Yaskawa INFORM job: DEMO_ROOF_SIDE_0625_3PAINT_39.JBI

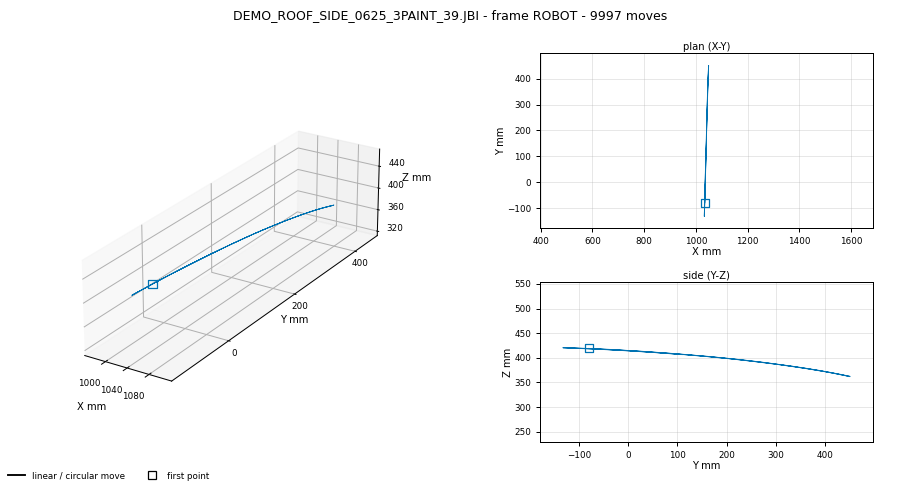
[picture p0: tool path of DEMO_ROOF_SIDE_0625_3PAINT_39.JBI in frame ROBOT, 9997 of 9997 moves have a stored position in this frame; points joined in program order, loops and branches not executed]
/JOB
//NAME DEMO_ROOF_SIDE_0625_3PAINT39
//POS
///NPOS 9997,0,0,0,0,0
///TOOL 0
///USER 0
///POSTYPE ROBOT
///RECTAN
///RCONF 1,0,0,0,0,0,0,0,0,0,0,0,0,0,0,0,0,0,0,0,0,0,0,0
C00000=1034.814,-80.144,419.319,168.128,39.375,157.359
C00001=1034.820,-79.894,419.308,168.131,39.374,157.359
C00002=1034.826,-79.644,419.297,168.134,39.373,157.359
C00003=1034.832,-79.394,419.285,168.136,39.372,157.359
C00004=1034.838,-79.144,419.275,168.139,39.372,157.359
C00005=1034.844,-78.895,419.264,168.142,39.371,157.359
C00006=1034.851,-78.645,419.253,168.144,39.371,157.359
C00007=1034.856,-78.396,419.242,168.147,39.370,157.358
C00008=1034.863,-78.145,419.231,168.150,39.369,157.358
C00009=1034.868,-77.896,419.220,168.152,39.368,157.358
C00010=1034.875,-77.646,419.209,168.155,39.368,157.358
C00011=1034.881,-77.397,419.197,168.157,39.367,157.358
C00012=1034.886,-77.147,419.186,168.160,39.366,157.358
C00013=1034.893,-76.897,419.175,168.162,39.365,157.358
C00014=1034.899,-76.648,419.164,168.165,39.364,157.358
C00015=1034.906,-76.398,419.154,168.168,39.364,157.358
C00016=1034.911,-76.148,419.143,168.170,39.363,157.358
C00017=1034.918,-75.899,419.131,168.173,39.362,157.358
C00018=1034.924,-75.649,419.120,168.176,39.361,157.358
C00019=1034.930,-75.399,419.109,168.179,39.361,157.358
C00020=1034.936,-75.150,419.098,168.181,39.360,157.358
C00021=1034.942,-74.899,419.086,168.184,39.360,157.358
C00022=1034.948,-74.650,419.075,168.187,39.359,157.358
C00023=1034.955,-74.400,419.064,168.189,39.358,157.358
C00024=1034.960,-74.151,419.053,168.192,39.358,157.358
C00025=1034.967,-73.901,419.041,168.195,39.357,157.358
C00026=1034.973,-73.652,419.030,168.196,39.356,157.358
C00027=1034.979,-73.402,419.019,168.199,39.356,157.358
C00028=1034.985,-73.153,419.007,168.202,39.355,157.358
C00029=1034.991,-72.902,418.995,168.204,39.355,157.358
C00030=1034.996,-72.653,418.984,168.207,39.354,157.358
C00031=1035.002,-72.404,418.973,168.210,39.354,157.358
C00032=1035.009,-72.154,418.962,168.212,39.353,157.358
C00033=1035.015,-71.904,418.951,168.215,39.352,157.358
C00034=1035.020,-71.654,418.938,168.217,39.352,157.358
C00035=1035.027,-71.404,418.927,168.220,39.351,157.358
C00036=1035.033,-71.155,418.915,168.223,39.351,157.358
C00037=1035.039,-70.905,418.904,168.225,39.350,157.358
C00038=1035.045,-70.656,418.893,168.228,39.350,157.358
C00039=1035.051,-70.406,418.881,168.231,39.349,157.358
C00040=1035.057,-70.156,418.870,168.233,39.348,157.357
C00041=1035.063,-69.907,418.858,168.236,39.348,157.357
C00042=1035.069,-69.657,418.847,168.239,39.347,157.357
C00043=1035.076,-69.408,418.835,168.241,39.347,157.357
C00044=1035.081,-69.158,418.823,168.244,39.346,157.357
C00045=1035.087,-68.908,418.812,168.246,39.346,157.357
C00046=1035.094,-68.658,418.800,168.249,39.345,157.357
C00047=1035.100,-68.375,418.787,168.251,39.344,157.357
C00048=1035.107,-68.093,418.774,168.254,39.344,157.357
C00049=1035.114,-67.811,418.761,168.257,39.343,157.357
C00050=1035.121,-67.528,418.748,168.260,39.342,157.357
C00051=1035.127,-67.278,418.736,168.263,39.342,157.357
C00052=1035.133,-67.028,418.724,168.265,39.341,157.357
C00053=1035.139,-66.778,418.713,168.268,39.341,157.357
C00054=1035.145,-66.529,418.701,168.271,39.340,157.357
C00055=1035.152,-66.279,418.690,168.273,39.340,157.357
C00056=1035.157,-66.029,418.677,168.276,39.339,157.357
C00057=1035.164,-65.780,418.666,168.278,39.339,157.357
C00058=1035.170,-65.530,418.655,168.281,39.338,157.357
C00059=1035.176,-65.281,418.643,168.284,39.337,157.357
C00060=1035.182,-65.030,418.631,168.286,39.337,157.357
C00061=1035.188,-64.781,418.619,168.289,39.336,157.357
C00062=1035.194,-64.532,418.607,168.292,39.336,157.357
C00063=1035.201,-64.282,418.596,168.294,39.335,157.357
C00064=1035.206,-64.032,418.584,168.297,39.335,157.357
C00065=1035.213,-63.783,418.572,168.299,39.334,157.357
C00066=1035.219,-63.533,418.561,168.302,39.334,157.357
C00067=1035.226,-63.283,418.549,168.305,39.333,157.357
C00068=1035.231,-63.034,418.537,168.307,39.333,157.357
C00069=1035.237,-62.784,418.525,168.310,39.332,157.357
C00070=1035.244,-62.534,418.513,168.311,39.331,157.357
C00071=1035.250,-62.285,418.502,168.314,39.331,157.357
C00072=1035.256,-62.035,418.489,168.317,39.330,157.357
C00073=1035.262,-61.785,418.478,168.319,39.330,157.357
C00074=1035.269,-61.536,418.466,168.322,39.329,157.357
C00075=1035.274,-61.286,418.454,168.324,39.329,157.357
C00076=1035.281,-61.037,418.442,168.327,39.328,157.357
C00077=1035.287,-60.787,418.431,168.330,39.327,157.357
C00078=1035.294,-60.537,418.419,168.332,39.327,157.357
C00079=1035.299,-60.288,418.406,168.335,39.326,157.357
C00080=1035.306,-60.038,418.394,168.338,39.326,157.357
C00081=1035.312,-59.788,418.383,168.340,39.325,157.357
C00082=1035.318,-59.538,418.371,168.343,39.325,157.357
C00083=1035.325,-59.289,418.359,168.345,39.324,157.357
C00084=1035.331,-59.040,418.347,168.348,39.324,157.357
C00085=1035.337,-58.790,418.335,168.351,39.323,157.357
C00086=1035.343,-58.540,418.323,168.353,39.322,157.357
C00087=1035.350,-58.290,418.311,168.356,39.322,157.357
C00088=1035.356,-58.041,418.299,168.358,39.321,157.357
C00089=1035.362,-57.791,418.287,168.361,39.321,157.357
C00090=1035.368,-57.542,418.275,168.364,39.320,157.357
C00091=1035.375,-57.292,418.263,168.366,39.320,157.357
C00092=1035.381,-57.042,418.251,168.369,39.319,157.357
C00093=1035.388,-56.793,418.239,168.371,39.319,157.357
C00094=1035.394,-56.543,418.227,168.374,39.318,157.357
C00095=1035.401,-56.294,418.215,168.375,39.318,157.357
C00096=1035.406,-56.044,418.203,168.378,39.317,157.357
C00097=1035.412,-55.794,418.191,168.381,39.316,157.357
C00098=1035.419,-55.545,418.179,168.383,39.316,157.357
C00099=1035.425,-55.295,418.167,168.386,39.315,157.357
C00100=1035.432,-55.045,418.155,168.388,39.315,157.357
C00101=1035.438,-54.796,418.143,168.391,39.314,157.357
C00102=1035.444,-54.546,418.130,168.394,39.313,157.357
C00103=1035.451,-54.296,418.118,168.396,39.313,157.357
C00104=1035.458,-54.047,418.107,168.399,39.312,157.357
C00105=1035.463,-53.797,418.094,168.401,39.312,157.357
C00106=1035.469,-53.548,418.082,168.404,39.311,157.356
C00107=1035.476,-53.298,418.070,168.407,39.311,157.357
C00108=1035.482,-53.048,418.058,168.409,39.310,157.356
C00109=1035.489,-52.799,418.046,168.412,39.310,157.357
C00110=1035.495,-52.549,418.034,168.414,39.309,157.356
C00111=1035.503,-52.268,418.020,168.417,39.309,157.356
C00112=1035.510,-51.986,418.006,168.420,39.308,157.356
C00113=1035.516,-51.705,417.992,168.423,39.307,157.356
C00114=1035.524,-51.423,417.979,168.426,39.307,157.356
C00115=1035.530,-51.174,417.966,168.428,39.306,157.356
C00116=1035.537,-50.924,417.954,168.431,39.306,157.356
C00117=1035.543,-50.674,417.942,168.434,39.305,157.356
C00118=1035.549,-50.424,417.930,168.436,39.305,157.356
C00119=1035.556,-50.175,417.916,168.439,39.305,157.356
C00120=1035.562,-49.926,417.904,168.440,39.304,157.356
C00121=1035.568,-49.676,417.892,168.444,39.304,157.356
C00122=1035.574,-49.426,417.879,168.446,39.304,157.356
C00123=1035.581,-49.176,417.867,168.449,39.304,157.357
C00124=1035.587,-48.927,417.854,168.450,39.303,157.356
C00125=1035.593,-48.677,417.841,168.453,39.303,157.356
C00126=1035.598,-48.428,417.829,168.456,39.302,157.357
C00127=1035.605,-48.178,417.817,168.459,39.302,157.357
C00128=1035.611,-47.929,417.804,168.460,39.301,157.356
C00129=1035.617,-47.679,417.792,168.463,39.301,157.357
C00130=1035.624,-47.430,417.780,168.465,39.301,157.357
C00131=1035.630,-47.180,417.766,168.468,39.300,157.357
C00132=1035.636,-46.931,417.754,168.470,39.300,157.357
C00133=1035.642,-46.681,417.741,168.473,39.300,157.357
C00134=1035.649,-46.432,417.729,168.475,39.300,157.357
C00135=1035.654,-46.182,417.716,168.478,39.299,157.357
C00136=1035.660,-45.932,417.703,168.480,39.299,157.357
C00137=1035.667,-45.683,417.690,168.483,39.298,157.357
C00138=1035.673,-45.433,417.678,168.485,39.298,157.357
C00139=1035.679,-45.183,417.666,168.488,39.297,157.357
C00140=1035.686,-44.933,417.652,168.490,39.297,157.357
C00141=1035.693,-44.684,417.640,168.493,39.297,157.357
C00142=1035.698,-44.434,417.627,168.495,39.297,157.357
C00143=1035.705,-44.185,417.614,168.498,39.296,157.357
C00144=1035.711,-43.935,417.602,168.500,39.296,157.357
C00145=1035.718,-43.686,417.589,168.503,39.296,157.357
C00146=1035.723,-43.436,417.576,168.505,39.295,157.357
C00147=1035.729,-43.186,417.564,168.507,39.295,157.357
C00148=1035.736,-42.937,417.551,168.510,39.294,157.357
C00149=1035.742,-42.687,417.539,168.512,39.294,157.357
C00150=1035.748,-42.438,417.525,168.515,39.293,157.357
C00151=1035.754,-42.188,417.513,168.517,39.293,157.357
C00152=1035.761,-41.939,417.500,168.520,39.293,157.357
C00153=1035.768,-41.688,417.487,168.522,39.293,157.357
C00154=1035.774,-41.439,417.474,168.525,39.292,157.357
C00155=1035.780,-41.189,417.461,168.527,39.292,157.357
C00156=1035.786,-40.940,417.448,168.530,39.292,157.357
C00157=1035.793,-40.690,417.436,168.532,39.292,157.357
C00158=1035.799,-40.441,417.423,168.535,39.291,157.357
C00159=1035.805,-40.191,417.410,168.537,39.291,157.357
C00160=1035.812,-39.941,417.397,168.540,39.290,157.357
C00161=1035.818,-39.691,417.384,168.542,39.290,157.357
C00162=1035.825,-39.442,417.371,168.545,39.289,157.357
C00163=1035.831,-39.193,417.359,168.547,39.289,157.357
C00164=1035.837,-38.943,417.346,168.550,39.289,157.357
C00165=1035.843,-38.694,417.332,168.552,39.289,157.357
C00166=1035.849,-38.443,417.319,168.554,39.288,157.357
C00167=1035.856,-38.194,417.306,168.557,39.288,157.357
C00168=1035.862,-37.944,417.294,168.559,39.288,157.357
C00169=1035.868,-37.695,417.280,168.562,39.287,157.357
C00170=1035.874,-37.446,417.267,168.564,39.287,157.357
C00171=1035.880,-37.196,417.255,168.567,39.287,157.357
C00172=1035.886,-36.947,417.241,168.569,39.287,157.357
C00173=1035.893,-36.697,417.228,168.571,39.287,157.357
C00174=1035.899,-36.447,417.214,168.574,39.287,157.357
C00175=1035.906,-36.167,417.200,168.576,39.286,157.357
C00176=1035.913,-35.885,417.185,168.579,39.286,157.357
C00177=1035.920,-35.604,417.170,168.582,39.285,157.357
C00178=1035.928,-35.323,417.156,168.585,39.285,157.358
C00179=1035.934,-35.074,417.142,168.587,39.285,157.358
C00180=1035.940,-34.824,417.129,168.589,39.285,157.358
C00181=1035.946,-34.574,417.117,168.592,39.285,157.358
C00182=1035.952,-34.325,417.103,168.594,39.284,157.358
C00183=1035.959,-34.075,417.090,168.597,39.284,157.358
C00184=1035.964,-33.826,417.076,168.599,39.284,157.358
C00185=1035.971,-33.576,417.063,168.601,39.283,157.358
C00186=1035.977,-33.326,417.050,168.604,39.283,157.358
C00187=1035.983,-33.076,417.036,168.606,39.283,157.358
C00188=1035.990,-32.827,417.023,168.609,39.283,157.358
C00189=1035.996,-32.578,417.010,168.611,39.283,157.358
C00190=1036.002,-32.329,416.997,168.614,39.282,157.358
C00191=1036.008,-32.078,416.984,168.616,39.282,157.358
C00192=1036.015,-31.829,416.970,168.618,39.282,157.358
C00193=1036.021,-31.580,416.957,168.621,39.282,157.358
C00194=1036.028,-31.330,416.943,168.623,39.281,157.358
C00195=1036.034,-31.080,416.930,168.626,39.281,157.358
C00196=1036.040,-30.831,416.917,168.628,39.281,157.358
C00197=1036.046,-30.582,416.904,168.630,39.281,157.358
C00198=1036.053,-30.332,416.890,168.633,39.280,157.358
C00199=1036.059,-30.082,416.877,168.635,39.280,157.358
C00200=1036.065,-29.833,416.864,168.637,39.280,157.358
C00201=1036.072,-29.583,416.851,168.640,39.280,157.358
C00202=1036.078,-29.333,416.837,168.643,39.280,157.358
C00203=1036.084,-29.084,416.823,168.645,39.279,157.358
C00204=1036.091,-28.834,416.810,168.647,39.279,157.358
C00205=1036.097,-28.585,416.797,168.649,39.279,157.358
C00206=1036.103,-28.335,416.783,168.652,39.278,157.358
C00207=1036.110,-28.085,416.770,168.654,39.278,157.358
C00208=1036.116,-27.836,416.756,168.658,39.278,157.359
C00209=1036.123,-27.586,416.743,168.660,39.278,157.359
C00210=1036.129,-27.337,416.729,168.662,39.278,157.359
C00211=1036.135,-27.088,416.716,168.665,39.277,157.359
C00212=1036.142,-26.838,416.703,168.667,39.277,157.359
C00213=1036.148,-26.588,416.689,168.669,39.277,157.359
C00214=1036.154,-26.339,416.675,168.672,39.277,157.359
C00215=1036.161,-26.089,416.662,168.674,39.277,157.359
C00216=1036.166,-25.839,416.648,168.676,39.277,157.359
C00217=1036.172,-25.590,416.635,168.679,39.276,157.359
C00218=1036.179,-25.341,416.620,168.681,39.276,157.359
C00219=1036.185,-25.091,416.606,168.683,39.276,157.359
C00220=1036.192,-24.841,416.593,168.686,39.276,157.359
C00221=1036.198,-24.592,416.580,168.688,39.276,157.359
C00222=1036.203,-24.342,416.566,168.690,39.276,157.359
C00223=1036.210,-24.092,416.552,168.693,39.275,157.359
C00224=1036.216,-23.843,416.539,168.695,39.275,157.359
C00225=1036.223,-23.593,416.524,168.697,39.275,157.359
C00226=1036.229,-23.344,416.511,168.700,39.275,157.359
C00227=1036.235,-23.095,416.497,168.702,39.275,157.359
C00228=1036.241,-22.845,416.483,168.704,39.275,157.359
C00229=1036.248,-22.595,416.470,168.707,39.274,157.359
C00230=1036.255,-22.346,416.455,168.709,39.274,157.359
C00231=1036.264,-21.949,416.434,168.713,39.275,157.360
C00232=1036.274,-21.552,416.412,168.716,39.274,157.360
C00233=1036.284,-21.155,416.389,168.720,39.274,157.360
C00234=1036.294,-20.758,416.368,168.724,39.274,157.360
C00235=1036.304,-20.374,416.346,168.727,39.274,157.360
C00236=1036.314,-19.990,416.325,168.731,39.273,157.360
C00237=1036.323,-19.606,416.304,168.735,39.273,157.360
C00238=1036.333,-19.222,416.282,168.738,39.273,157.360
C00239=1036.339,-18.973,416.268,168.740,39.273,157.360
C00240=1036.346,-18.723,416.255,168.743,39.272,157.360
C00241=1036.352,-18.474,416.241,168.745,39.272,157.360
C00242=1036.358,-18.224,416.227,168.747,39.272,157.360
C00243=1036.365,-17.975,416.213,168.750,39.272,157.360
C00244=1036.371,-17.725,416.198,168.753,39.272,157.360
C00245=1036.377,-17.476,416.185,168.755,39.272,157.360
C00246=1036.384,-17.226,416.171,168.758,39.271,157.360
C00247=1036.390,-16.977,416.157,168.760,39.271,157.361
C00248=1036.397,-16.727,416.143,168.762,39.271,157.361
C00249=1036.403,-16.477,416.128,168.765,39.271,157.361
C00250=1036.409,-16.228,416.115,168.767,39.271,157.361
C00251=1036.416,-15.979,416.101,168.769,39.271,157.361
C00252=1036.422,-15.729,416.087,168.771,39.271,157.361
C00253=1036.429,-15.479,416.073,168.774,39.270,157.361
C00254=1036.434,-15.230,416.059,168.776,39.270,157.361
C00255=1036.441,-14.980,416.045,168.778,39.271,157.361
C00256=1036.447,-14.731,416.030,168.781,39.270,157.361
C00257=1036.454,-14.481,416.017,168.783,39.270,157.361
C00258=1036.460,-14.231,416.002,168.785,39.270,157.361
C00259=1036.466,-13.982,415.988,168.787,39.270,157.361
C00260=1036.473,-13.733,415.974,168.790,39.270,157.361
C00261=1036.478,-13.483,415.960,168.792,39.270,157.361
C00262=1036.485,-13.233,415.945,168.794,39.270,157.361
C00263=1036.491,-12.985,415.931,168.796,39.270,157.361
C00264=1036.497,-12.734,415.917,168.799,39.270,157.361
C00265=1036.504,-12.485,415.902,168.801,39.270,157.362
C00266=1036.510,-12.235,415.888,168.803,39.270,157.362
C00267=1036.516,-11.986,415.873,168.805,39.270,157.362
C00268=1036.522,-11.737,415.860,168.808,39.270,157.362
C00269=1036.529,-11.487,415.845,168.810,39.270,157.362
C00270=1036.535,-11.237,415.830,168.812,39.270,157.362
C00271=1036.541,-10.988,415.817,168.814,39.269,157.362
C00272=1036.548,-10.738,415.802,168.818,39.270,157.362
C00273=1036.554,-10.489,415.787,168.820,39.270,157.362
C00274=1036.560,-10.239,415.774,168.822,39.270,157.362
C00275=1036.567,-9.990,415.759,168.824,39.269,157.362
C00276=1036.573,-9.741,415.744,168.827,39.269,157.362
C00277=1036.579,-9.491,415.731,168.829,39.269,157.362
C00278=1036.586,-9.241,415.716,168.831,39.270,157.362
C00279=1036.592,-8.992,415.701,168.833,39.269,157.362
C00280=1036.598,-8.742,415.688,168.836,39.269,157.362
C00281=1036.605,-8.493,415.673,168.838,39.269,157.363
C00282=1036.611,-8.244,415.658,168.840,39.269,157.363
C00283=1036.617,-7.994,415.644,168.842,39.269,157.363
C00284=1036.624,-7.744,415.629,168.844,39.269,157.363
C00285=1036.630,-7.495,415.615,168.847,39.269,157.363
C00286=1036.637,-7.246,415.600,168.849,39.269,157.363
C00287=1036.643,-6.995,415.586,168.851,39.269,157.363
C00288=1036.648,-6.746,415.572,168.853,39.269,157.363
C00289=1036.656,-6.497,415.557,168.856,39.268,157.363
C00290=1036.662,-6.247,415.542,168.858,39.268,157.363
C00291=1036.668,-5.997,415.528,168.860,39.269,157.363
C00292=1036.675,-5.749,415.514,168.862,39.269,157.363
C00293=1036.681,-5.499,415.499,168.865,39.268,157.363
C00294=1036.687,-5.249,415.484,168.867,39.268,157.363
C00295=1036.694,-5.001,415.470,168.869,39.268,157.363
C00296=1036.700,-4.750,415.456,168.871,39.268,157.363
C00297=1036.706,-4.501,415.441,168.873,39.268,157.363
C00298=1036.713,-4.251,415.427,168.877,39.268,157.364
C00299=1036.721,-3.968,415.410,168.879,39.268,157.364
C00300=1036.728,-3.685,415.393,168.882,39.268,157.364
C00301=1036.734,-3.401,415.376,168.884,39.268,157.364
C00302=1036.741,-3.118,415.360,168.887,39.268,157.364
C00303=1036.748,-2.868,415.345,168.889,39.268,157.364
C00304=1036.754,-2.618,415.330,168.891,39.268,157.364
C00305=1036.760,-2.369,415.315,168.893,39.268,157.364
C00306=1036.766,-2.120,415.301,168.895,39.268,157.364
C00307=1036.773,-1.870,415.286,168.898,39.268,157.364
C00308=1036.779,-1.620,415.271,168.900,39.269,157.364
C00309=1036.785,-1.372,415.256,168.902,39.268,157.364
C00310=1036.791,-1.122,415.241,168.904,39.268,157.364
C00311=1036.798,-0.872,415.226,168.906,39.269,157.365
C00312=1036.804,-0.623,415.211,168.908,39.269,157.365
C00313=1036.810,-0.373,415.196,168.911,39.268,157.365
C00314=1036.816,-0.124,415.182,168.914,39.269,157.365
C00315=1036.823,0.126,415.167,168.916,39.269,157.365
C00316=1036.829,0.375,415.152,168.918,39.269,157.365
C00317=1036.835,0.625,415.137,168.920,39.269,157.365
C00318=1036.841,0.874,415.122,168.922,39.269,157.365
C00319=1036.847,1.124,415.107,168.924,39.269,157.365
C00320=1036.854,1.373,415.092,168.927,39.269,157.365
C00321=1036.860,1.623,415.078,168.929,39.269,157.365
C00322=1036.867,1.872,415.062,168.931,39.269,157.365
C00323=1036.873,2.121,415.047,168.933,39.270,157.366
C00324=1036.879,2.371,415.032,168.935,39.269,157.366
C00325=1036.885,2.620,415.017,168.937,39.269,157.366
C00326=1036.892,2.870,415.002,168.940,39.270,157.366
C00327=1036.898,3.120,414.987,168.942,39.270,157.366
C00328=1036.904,3.370,414.972,168.944,39.269,157.366
C00329=1036.910,3.619,414.957,168.946,39.270,157.366
C00330=1036.916,3.868,414.942,168.948,39.270,157.366
C00331=1036.923,4.117,414.927,168.950,39.270,157.366
C00332=1036.929,4.367,414.912,168.953,39.270,157.366
C00333=1036.935,4.617,414.897,168.956,39.270,157.366
C00334=1036.942,4.866,414.882,168.958,39.270,157.366
C00335=1036.948,5.116,414.867,168.960,39.270,157.366
C00336=1036.954,5.364,414.852,168.962,39.270,157.367
C00337=1036.961,5.614,414.837,168.964,39.270,157.367
C00338=1036.967,5.863,414.822,168.966,39.270,157.367
C00339=1036.973,6.113,414.807,168.969,39.270,157.367
C00340=1036.980,6.362,414.791,168.971,39.270,157.367
C00341=1036.987,6.612,414.776,168.973,39.270,157.367
C00342=1036.993,6.861,414.761,168.975,39.270,157.367
C00343=1036.999,7.111,414.746,168.977,39.270,157.367
C00344=1037.006,7.360,414.731,168.979,39.270,157.367
C00345=1037.012,7.610,414.716,168.981,39.270,157.367
C00346=1037.018,7.860,414.700,168.984,39.270,157.367
C00347=1037.024,8.109,414.686,168.986,39.270,157.367
C00348=1037.031,8.358,414.670,168.988,39.270,157.367
C00349=1037.037,8.607,414.655,168.991,39.271,157.368
C00350=1037.043,8.857,414.640,168.993,39.271,157.368
C00351=1037.050,9.106,414.624,168.995,39.270,157.368
C00352=1037.056,9.356,414.609,168.997,39.270,157.368
C00353=1037.063,9.605,414.595,169.000,39.271,157.368
C00354=1037.069,9.854,414.579,169.002,39.271,157.368
C00355=1037.076,10.104,414.564,169.004,39.270,157.368
C00356=1037.082,10.354,414.549,169.006,39.271,157.368
C00357=1037.089,10.603,414.533,169.008,39.271,157.368
C00358=1037.095,10.853,414.518,169.010,39.271,157.368
C00359=1037.101,11.102,414.503,169.012,39.270,157.368
C00360=1037.108,11.352,414.487,169.014,39.271,157.368
C00361=1037.114,11.601,414.472,169.017,39.271,157.368
C00362=1037.120,11.851,414.457,169.019,39.271,157.368
C00363=1037.128,12.136,414.440,169.021,39.271,157.369
C00364=1037.135,12.421,414.422,169.024,39.271,157.369
C00365=1037.143,12.706,414.404,169.026,39.271,157.369
C00366=1037.150,12.992,414.387,169.029,39.271,157.369
C00367=1037.157,13.241,414.372,169.032,39.271,157.369
C00368=1037.163,13.491,414.357,169.034,39.271,157.369
C00369=1037.170,13.740,414.341,169.036,39.271,157.369
C00370=1037.176,13.990,414.325,169.038,39.271,157.369
C00371=1037.182,14.239,414.310,169.040,39.271,157.369
C00372=1037.189,14.489,414.295,169.042,39.271,157.369
C00373=1037.195,14.738,414.279,169.044,39.271,157.369
C00374=1037.201,14.988,414.264,169.046,39.271,157.369
C00375=1037.208,15.237,414.248,169.048,39.272,157.370
C00376=1037.214,15.486,414.232,169.051,39.272,157.370
C00377=1037.220,15.736,414.217,169.053,39.271,157.370
C00378=1037.227,15.985,414.201,169.055,39.272,157.370
C00379=1037.232,16.235,414.186,169.057,39.272,157.370
C00380=1037.239,16.484,414.170,169.059,39.272,157.370
C00381=1037.245,16.734,414.154,169.061,39.272,157.370
C00382=1037.251,16.983,414.139,169.063,39.272,157.370
C00383=1037.258,17.232,414.123,169.066,39.273,157.370
C00384=1037.264,17.482,414.107,169.068,39.272,157.370
C00385=1037.271,17.732,414.091,169.070,39.273,157.370
C00386=1037.278,17.981,414.076,169.072,39.273,157.371
C00387=1037.283,18.231,414.060,169.074,39.273,157.371
C00388=1037.290,18.480,414.045,169.077,39.273,157.371
C00389=1037.297,18.729,414.029,169.079,39.273,157.371
C00390=1037.302,18.979,414.013,169.081,39.273,157.371
C00391=1037.309,19.228,413.998,169.083,39.273,157.371
C00392=1037.315,19.477,413.981,169.085,39.273,157.371
C00393=1037.321,19.727,413.967,169.087,39.274,157.371
C00394=1037.328,19.976,413.951,169.089,39.273,157.371
C00395=1037.335,20.226,413.934,169.091,39.274,157.371
C00396=1037.341,20.475,413.919,169.093,39.274,157.371
C00397=1037.347,20.725,413.903,169.095,39.274,157.371
C00398=1037.354,20.974,413.887,169.098,39.274,157.372
C00399=1037.360,21.223,413.871,169.100,39.274,157.372
C00400=1037.366,21.473,413.856,169.102,39.275,157.372
C00401=1037.372,21.722,413.840,169.104,39.274,157.372
C00402=1037.378,21.971,413.824,169.106,39.275,157.372
C00403=1037.385,22.221,413.808,169.109,39.275,157.372
C00404=1037.391,22.471,413.791,169.111,39.275,157.372
C00405=1037.398,22.720,413.776,169.113,39.275,157.372
C00406=1037.403,22.970,413.760,169.115,39.276,157.372
C00407=1037.410,23.219,413.745,169.117,39.275,157.372
C00408=1037.416,23.468,413.728,169.119,39.275,157.372
C00409=1037.423,23.717,413.713,169.121,39.276,157.373
C00410=1037.429,23.966,413.696,169.123,39.276,157.373
C00411=1037.436,24.217,413.681,169.126,39.276,157.373
C00412=1037.442,24.466,413.665,169.128,39.276,157.373
C00413=1037.448,24.715,413.649,169.130,39.277,157.373
C00414=1037.454,24.964,413.633,169.132,39.276,157.373
C00415=1037.461,25.213,413.617,169.134,39.276,157.373
C00416=1037.467,25.463,413.601,169.136,39.277,157.373
C00417=1037.474,25.713,413.585,169.138,39.277,157.373
C00418=1037.480,25.962,413.569,169.140,39.277,157.373
C00419=1037.486,26.211,413.552,169.142,39.277,157.373
C00420=1037.493,26.461,413.537,169.144,39.277,157.374
C00421=1037.499,26.711,413.521,169.146,39.277,157.374
C00422=1037.506,26.960,413.505,169.149,39.278,157.374
C00423=1037.512,27.209,413.489,169.151,39.278,157.374
C00424=1037.518,27.459,413.473,169.153,39.277,157.374
C00425=1037.524,27.708,413.457,169.156,39.278,157.374
C00426=1037.531,27.958,413.440,169.158,39.278,157.374
C00427=1037.538,28.244,413.422,169.160,39.278,157.374
C00428=1037.545,28.531,413.404,169.162,39.278,157.374
C00429=1037.553,28.817,413.385,169.165,39.279,157.374
C00430=1037.559,29.104,413.366,169.167,39.279,157.375
C00431=1037.567,29.353,413.350,169.169,39.279,157.375
C00432=1037.573,29.603,413.334,169.171,39.279,157.375
C00433=1037.579,29.852,413.317,169.173,39.279,157.375
C00434=1037.585,30.101,413.301,169.175,39.280,157.375
C00435=1037.592,30.351,413.285,169.177,39.280,157.375
C00436=1037.598,30.601,413.269,169.179,39.280,157.375
C00437=1037.604,30.850,413.253,169.182,39.280,157.375
C00438=1037.610,31.099,413.236,169.184,39.280,157.375
C00439=1037.616,31.348,413.219,169.186,39.280,157.375
C00440=1037.623,31.598,413.203,169.188,39.281,157.376
C00441=1037.629,31.847,413.187,169.190,39.281,157.376
C00442=1037.635,32.096,413.171,169.192,39.281,157.376
C00443=1037.642,32.346,413.154,169.194,39.281,157.376
C00444=1037.648,32.596,413.139,169.196,39.282,157.376
C00445=1037.654,32.845,413.122,169.198,39.281,157.376
C00446=1037.661,33.094,413.105,169.200,39.282,157.376
C00447=1037.667,33.344,413.089,169.202,39.282,157.376
C00448=1037.673,33.593,413.072,169.204,39.282,157.376
C00449=1037.680,33.842,413.057,169.207,39.283,157.377
C00450=1037.686,34.092,413.040,169.209,39.283,157.377
C00451=1037.693,34.341,413.023,169.211,39.283,157.377
C00452=1037.699,34.590,413.007,169.213,39.283,157.377
C00453=1037.706,34.840,412.991,169.215,39.283,157.377
C00454=1037.712,35.089,412.975,169.217,39.283,157.377
C00455=1037.718,35.339,412.958,169.219,39.283,157.377
C00456=1037.725,35.588,412.941,169.221,39.284,157.377
C00457=1037.731,35.837,412.925,169.223,39.284,157.377
C00458=1037.737,36.086,412.909,169.225,39.284,157.377
C00459=1037.744,36.336,412.892,169.227,39.284,157.377
C00460=1037.750,36.585,412.876,169.229,39.284,157.378
C00461=1037.756,36.835,412.859,169.231,39.284,157.378
C00462=1037.763,37.085,412.843,169.234,39.285,157.378
C00463=1037.769,37.333,412.826,169.236,39.285,157.378
C00464=1037.775,37.583,412.809,169.238,39.285,157.378
C00465=1037.781,37.833,412.793,169.240,39.286,157.378
C00466=1037.788,38.081,412.776,169.242,39.285,157.378
C00467=1037.794,38.332,412.759,169.244,39.286,157.378
C00468=1037.800,38.581,412.743,169.246,39.286,157.378
C00469=1037.806,38.830,412.726,169.248,39.286,157.379
C00470=1037.813,39.080,412.709,169.250,39.287,157.379
C00471=1037.819,39.329,412.693,169.252,39.287,157.379
C00472=1037.825,39.578,412.676,169.254,39.287,157.379
C00473=1037.832,39.828,412.659,169.257,39.287,157.379
C00474=1037.838,40.076,412.643,169.259,39.288,157.379
C00475=1037.844,40.326,412.626,169.261,39.287,157.379
C00476=1037.851,40.575,412.609,169.263,39.288,157.379
C00477=1037.857,40.825,412.593,169.265,39.288,157.379
C00478=1037.863,41.075,412.576,169.267,39.288,157.379
C00479=1037.870,41.323,412.559,169.269,39.289,157.380
C00480=1037.875,41.573,412.543,169.271,39.289,157.380
C00481=1037.882,41.822,412.525,169.273,39.289,157.380
C00482=1037.888,42.072,412.509,169.275,39.290,157.380
C00483=1037.895,42.321,412.492,169.277,39.289,157.380
C00484=1037.901,42.570,412.476,169.280,39.290,157.380
C00485=1037.907,42.819,412.459,169.282,39.290,157.380
C00486=1037.914,43.069,412.442,169.284,39.290,157.380
C00487=1037.920,43.318,412.425,169.286,39.290,157.380
C00488=1037.926,43.568,412.408,169.288,39.291,157.381
C00489=1037.932,43.817,412.391,169.290,39.291,157.381
C00490=1037.939,44.067,412.374,169.292,39.292,157.381
C00491=1037.946,44.353,412.354,169.294,39.291,157.381
C00492=1037.952,44.639,412.335,169.296,39.292,157.381
C00493=1037.960,44.926,412.315,169.298,39.292,157.381
C00494=1037.967,45.213,412.296,169.302,39.293,157.381
C00495=1037.973,45.461,412.279,169.304,39.293,157.382
C00496=1037.979,45.711,412.262,169.305,39.293,157.382
C00497=1037.985,45.960,412.244,169.307,39.294,157.382
C00498=1037.992,46.210,412.227,169.309,39.294,157.382
C00499=1037.998,46.459,412.211,169.311,39.294,157.382
C00500=1038.005,46.709,412.193,169.313,39.295,157.382
C00501=1038.010,46.958,412.176,169.315,39.295,157.382
C00502=1038.016,47.207,412.160,169.317,39.295,157.382
C00503=1038.023,47.456,412.142,169.320,39.296,157.382
C00504=1038.028,47.706,412.125,169.322,39.296,157.383
C00505=1038.035,47.956,412.108,169.324,39.296,157.383
C00506=1038.041,48.204,412.091,169.326,39.296,157.383
C00507=1038.047,48.454,412.073,169.328,39.297,157.383
C00508=1038.054,48.703,412.056,169.330,39.297,157.383
C00509=1038.060,48.953,412.040,169.332,39.297,157.383
C00510=1038.066,49.202,412.022,169.334,39.298,157.383
C00511=1038.073,49.451,412.005,169.336,39.298,157.384
C00512=1038.079,49.701,411.988,169.337,39.298,157.384
C00513=1038.085,49.950,411.970,169.340,39.299,157.384
C00514=1038.091,50.199,411.953,169.342,39.299,157.384
C00515=1038.098,50.449,411.936,169.344,39.299,157.384
C00516=1038.104,50.697,411.919,169.346,39.300,157.384
C00517=1038.110,50.948,411.902,169.348,39.300,157.384
C00518=1038.116,51.196,411.885,169.350,39.300,157.384
C00519=1038.123,51.446,411.868,169.352,39.300,157.384
C00520=1038.128,51.695,411.850,169.354,39.300,157.384
C00521=1038.135,51.944,411.833,169.356,39.301,157.385
C00522=1038.142,52.194,411.816,169.358,39.301,157.385
C00523=1038.147,52.443,411.799,169.360,39.301,157.385
C00524=1038.154,52.693,411.781,169.363,39.302,157.385
C00525=1038.161,52.942,411.764,169.365,39.302,157.385
C00526=1038.167,53.191,411.746,169.367,39.302,157.385
C00527=1038.173,53.440,411.729,169.369,39.302,157.385
C00528=1038.179,53.690,411.711,169.371,39.303,157.385
C00529=1038.185,53.939,411.695,169.373,39.303,157.386
C00530=1038.192,54.189,411.678,169.375,39.303,157.386
C00531=1038.198,54.438,411.660,169.376,39.304,157.386
C00532=1038.204,54.687,411.643,169.378,39.304,157.386
C00533=1038.211,54.936,411.626,169.381,39.304,157.386
C00534=1038.217,55.185,411.608,169.383,39.304,157.386
C00535=1038.223,55.435,411.591,169.385,39.305,157.386
C00536=1038.230,55.684,411.573,169.387,39.305,157.386
C00537=1038.236,55.933,411.556,169.389,39.305,157.386
C00538=1038.243,56.183,411.538,169.391,39.305,157.387
C00539=1038.250,56.432,411.521,169.393,39.305,157.387
C00540=1038.255,56.681,411.504,169.395,39.306,157.387
C00541=1038.262,56.931,411.486,169.397,39.306,157.387
C00542=1038.267,57.180,411.469,169.399,39.306,157.387
C00543=1038.274,57.429,411.451,169.401,39.307,157.387
C00544=1038.281,57.679,411.435,169.404,39.307,157.387
C00545=1038.286,57.928,411.417,169.406,39.307,157.387
C00546=1038.293,58.178,411.400,169.408,39.307,157.387
C00547=1038.300,58.427,411.382,169.410,39.307,157.388
C00548=1038.306,58.676,411.364,169.412,39.308,157.388
C00549=1038.313,58.925,411.347,169.414,39.308,157.388
C00550=1038.320,59.174,411.329,169.416,39.308,157.388
C00551=1038.325,59.423,411.312,169.418,39.309,157.388
C00552=1038.332,59.673,411.295,169.419,39.309,157.388
C00553=1038.338,59.923,411.277,169.421,39.309,157.388
C00554=1038.345,60.172,411.259,169.423,39.309,157.388
C00555=1038.352,60.458,411.239,169.427,39.309,157.388
C00556=1038.360,60.745,411.219,169.429,39.310,157.389
C00557=1038.366,61.031,411.199,169.431,39.310,157.389
C00558=1038.374,61.317,411.179,169.433,39.310,157.389
C00559=1038.380,61.566,411.162,169.435,39.311,157.389
C00560=1038.387,61.815,411.144,169.437,39.310,157.389
C00561=1038.393,62.065,411.126,169.439,39.311,157.389
C00562=1038.400,62.315,411.109,169.441,39.311,157.389
C00563=1038.406,62.564,411.092,169.443,39.311,157.389
C00564=1038.413,62.812,411.074,169.445,39.311,157.389
C00565=1038.420,63.062,411.056,169.447,39.312,157.390
C00566=1038.426,63.312,411.038,169.450,39.312,157.390
C00567=1038.432,63.560,411.021,169.452,39.312,157.390
C00568=1038.438,63.810,411.003,169.454,39.312,157.390
C00569=1038.445,64.059,410.986,169.456,39.312,157.390
C00570=1038.451,64.309,410.967,169.458,39.313,157.390
C00571=1038.457,64.558,410.950,169.460,39.313,157.390
C00572=1038.464,64.807,410.932,169.462,39.314,157.390
C00573=1038.470,65.057,410.915,169.464,39.314,157.390
C00574=1038.476,65.306,410.896,169.466,39.314,157.391
C00575=1038.483,65.555,410.879,169.468,39.315,157.391
C00576=1038.489,65.804,410.861,169.470,39.315,157.391
C00577=1038.495,66.053,410.842,169.472,39.315,157.391
C00578=1038.502,66.303,410.825,169.474,39.316,157.391
C00579=1038.508,66.552,410.807,169.476,39.315,157.391
C00580=1038.514,66.802,410.789,169.478,39.316,157.391
C00581=1038.521,67.050,410.771,169.480,39.316,157.391
C00582=1038.527,67.300,410.754,169.482,39.317,157.392
C00583=1038.532,67.549,410.736,169.484,39.317,157.392
C00584=1038.539,67.798,410.717,169.486,39.317,157.392
C00585=1038.546,68.048,410.700,169.489,39.318,157.392
C00586=1038.552,68.297,410.681,169.491,39.318,157.392
C00587=1038.558,68.546,410.664,169.493,39.318,157.392
C00588=1038.565,68.795,410.646,169.494,39.319,157.392
C00589=1038.571,69.045,410.628,169.496,39.319,157.393
C00590=1038.577,69.294,410.610,169.498,39.319,157.393
C00591=1038.584,69.543,410.591,169.500,39.320,157.393
C00592=1038.589,69.792,410.574,169.502,39.320,157.393
C00593=1038.596,70.042,410.556,169.504,39.320,157.393
C00594=1038.602,70.291,410.538,169.506,39.320,157.393
C00595=1038.608,70.541,410.520,169.509,39.321,157.393
C00596=1038.615,70.790,410.501,169.511,39.321,157.393
C00597=1038.620,71.039,410.483,169.513,39.322,157.394
C00598=1038.627,71.288,410.465,169.515,39.322,157.394
C00599=1038.633,71.538,410.447,169.517,39.322,157.394
C00600=1038.640,71.787,410.429,169.518,39.323,157.394
C00601=1038.646,72.036,410.411,169.520,39.323,157.394
C00602=1038.652,72.285,410.393,169.522,39.323,157.394
C00603=1038.658,72.534,410.375,169.524,39.324,157.394
C00604=1038.665,72.784,410.356,169.527,39.324,157.394
C00605=1038.671,73.033,410.338,169.529,39.325,157.395
C00606=1038.677,73.282,410.319,169.531,39.324,157.395
C00607=1038.683,73.532,410.302,169.533,39.325,157.395
C00608=1038.689,73.781,410.283,169.535,39.325,157.395
C00609=1038.696,74.030,410.265,169.537,39.326,157.395
C00610=1038.702,74.279,410.247,169.539,39.326,157.395
C00611=1038.709,74.528,410.229,169.540,39.326,157.395
C00612=1038.715,74.778,410.211,169.543,39.327,157.395
C00613=1038.721,75.027,410.192,169.545,39.327,157.396
C00614=1038.728,75.276,410.173,169.547,39.327,157.396
C00615=1038.733,75.525,410.156,169.549,39.328,157.396
C00616=1038.740,75.774,410.137,169.551,39.328,157.396
C00617=1038.746,76.024,410.119,169.553,39.329,157.396
C00618=1038.752,76.273,410.101,169.555,39.328,157.396
C00619=1038.760,76.559,410.080,169.557,39.329,157.396
C00620=1038.767,76.845,410.058,169.559,39.329,157.396
C00621=1038.774,77.132,410.038,169.563,39.330,157.397
C00622=1038.781,77.418,410.016,169.565,39.330,157.397
C00623=1038.788,77.667,409.998,169.567,39.331,157.397
C00624=1038.794,77.915,409.979,169.569,39.331,157.397
C00625=1038.800,78.165,409.961,169.570,39.331,157.397
C00626=1038.806,78.414,409.943,169.572,39.332,157.397
C00627=1038.813,78.663,409.924,169.574,39.332,157.397
C00628=1038.819,78.913,409.906,169.576,39.333,157.398
C00629=1038.825,79.162,409.888,169.578,39.333,157.398
C00630=1038.831,79.412,409.868,169.581,39.333,157.398
C00631=1038.837,79.661,409.850,169.583,39.334,157.398
C00632=1038.844,79.910,409.831,169.585,39.334,157.398
C00633=1038.850,80.160,409.813,169.587,39.335,157.398
C00634=1038.856,80.408,409.795,169.589,39.335,157.398
C00635=1038.861,80.658,409.776,169.590,39.336,157.399
C00636=1038.868,80.907,409.757,169.592,39.335,157.399
C00637=1038.874,81.156,409.738,169.594,39.336,157.399
C00638=1038.881,81.405,409.720,169.597,39.336,157.399
C00639=1038.887,81.655,409.702,169.599,39.337,157.399
C00640=1038.893,81.904,409.683,169.601,39.337,157.399
C00641=1038.899,82.153,409.664,169.603,39.338,157.399
C00642=1038.905,82.402,409.645,169.605,39.338,157.400
C00643=1038.912,82.651,409.627,169.607,39.338,157.400
C00644=1038.918,82.901,409.608,169.609,39.339,157.400
C00645=1038.925,83.150,409.589,169.610,39.339,157.400
C00646=1038.930,83.399,409.570,169.613,39.340,157.400
C00647=1038.937,83.648,409.551,169.615,39.340,157.400
C00648=1038.943,83.898,409.533,169.617,39.340,157.400
C00649=1038.949,84.147,409.515,169.619,39.341,157.401
C00650=1038.956,84.396,409.496,169.621,39.341,157.401
C00651=1038.961,84.646,409.477,169.623,39.342,157.401
C00652=1038.968,84.895,409.458,169.625,39.342,157.401
C00653=1038.974,85.144,409.440,169.627,39.342,157.401
C00654=1038.981,85.393,409.421,169.630,39.342,157.401
C00655=1038.987,85.642,409.402,169.632,39.343,157.401
C00656=1038.993,85.892,409.383,169.634,39.343,157.402
C00657=1038.999,86.141,409.364,169.635,39.344,157.402
C00658=1039.006,86.390,409.346,169.637,39.344,157.402
C00659=1039.012,86.639,409.327,169.639,39.344,157.402
C00660=1039.018,86.888,409.308,169.641,39.345,157.402
C00661=1039.024,87.138,409.289,169.643,39.345,157.402
C00662=1039.031,87.387,409.271,169.646,39.346,157.402
C00663=1039.037,87.636,409.252,169.648,39.346,157.402
C00664=1039.043,87.885,409.233,169.650,39.346,157.403
C00665=1039.049,88.134,409.214,169.652,39.347,157.403
C00666=1039.055,88.383,409.195,169.654,39.347,157.403
C00667=1039.062,88.633,409.177,169.656,39.348,157.403
C00668=1039.068,88.882,409.158,169.658,39.347,157.403
C00669=1039.075,89.131,409.139,169.660,39.348,157.403
C00670=1039.080,89.380,409.120,169.661,39.348,157.403
C00671=1039.087,89.630,409.101,169.664,39.349,157.404
C00672=1039.094,89.879,409.082,169.666,39.349,157.404
C00673=1039.101,90.128,409.063,169.668,39.349,157.404
C00674=1039.106,90.377,409.044,169.670,39.350,157.404
C00675=1039.113,90.626,409.025,169.672,39.350,157.404
C00676=1039.118,90.876,409.006,169.674,39.351,157.404
C00677=1039.125,91.125,408.987,169.676,39.351,157.404
C00678=1039.131,91.374,408.967,169.678,39.352,157.405
C00679=1039.137,91.623,408.949,169.681,39.352,157.405
C00680=1039.143,91.872,408.929,169.683,39.353,157.405
C00681=1039.149,92.121,408.911,169.684,39.353,157.405
C00682=1039.155,92.371,408.892,169.686,39.353,157.405
C00683=1039.163,92.656,408.869,169.689,39.354,157.405
C00684=1039.170,92.943,408.848,169.691,39.355,157.406
C00685=1039.177,93.228,408.825,169.693,39.355,157.406
C00686=1039.184,93.515,408.804,169.696,39.356,157.406
C00687=1039.190,93.764,408.784,169.698,39.356,157.406
C00688=1039.197,94.013,408.765,169.700,39.356,157.406
C00689=1039.202,94.262,408.746,169.702,39.356,157.406
C00690=1039.209,94.511,408.727,169.704,39.357,157.406
C00691=1039.215,94.760,408.707,169.706,39.357,157.407
C00692=1039.221,95.009,408.689,169.708,39.358,157.407
C00693=1039.227,95.259,408.669,169.711,39.358,157.407
C00694=1039.234,95.508,408.650,169.712,39.359,157.407
C00695=1039.240,95.757,408.630,169.714,39.359,157.407
C00696=1039.246,96.007,408.611,169.716,39.359,157.407
C00697=1039.252,96.255,408.592,169.718,39.360,157.407
C00698=1039.258,96.505,408.572,169.720,39.360,157.408
C00699=1039.264,96.754,408.554,169.722,39.361,157.408
C00700=1039.271,97.003,408.534,169.724,39.361,157.408
C00701=1039.277,97.252,408.515,169.727,39.362,157.408
C00702=1039.283,97.502,408.496,169.729,39.362,157.408
C00703=1039.290,97.750,408.476,169.731,39.363,157.408
C00704=1039.296,98.000,408.457,169.733,39.363,157.408
C00705=1039.302,98.249,408.438,169.735,39.363,157.409
C00706=1039.309,98.498,408.418,169.737,39.364,157.409
C00707=1039.315,98.748,408.399,169.739,39.364,157.409
C00708=1039.321,98.996,408.379,169.740,39.365,157.409
C00709=1039.327,99.245,408.361,169.743,39.365,157.409
C00710=1039.333,99.494,408.341,169.745,39.366,157.409
C00711=1039.340,99.744,408.321,169.747,39.365,157.409
C00712=1039.346,99.994,408.303,169.749,39.366,157.410
C00713=1039.352,100.242,408.283,169.751,39.366,157.410
C00714=1039.359,100.491,408.264,169.753,39.367,157.410
C00715=1039.365,100.740,408.244,169.755,39.367,157.410
C00716=1039.371,100.990,408.224,169.757,39.368,157.410
C00717=1039.377,101.239,408.204,169.760,39.368,157.410
C00718=1039.384,101.488,408.185,169.762,39.369,157.410
C00719=1039.389,101.737,408.166,169.764,39.369,157.411
C00720=1039.395,101.986,408.146,169.766,39.370,157.411
C00721=1039.402,102.236,408.126,169.768,39.370,157.411
C00722=1039.408,102.485,408.106,169.769,39.371,157.411
C00723=1039.414,102.734,408.088,169.771,39.371,157.411
C00724=1039.420,102.983,408.068,169.774,39.372,157.411
C00725=1039.426,103.232,408.048,169.776,39.372,157.412
C00726=1039.432,103.482,408.028,169.778,39.373,157.412
C00727=1039.438,103.731,408.008,169.780,39.373,157.412
C00728=1039.445,103.979,407.989,169.782,39.374,157.412
C00729=1039.451,104.229,407.970,169.784,39.374,157.412
C00730=1039.457,104.478,407.949,169.786,39.375,157.412
C00731=1039.463,104.728,407.930,169.789,39.375,157.413
C00732=1039.469,104.976,407.910,169.791,39.376,157.413
C00733=1039.475,105.225,407.890,169.793,39.376,157.413
C00734=1039.482,105.475,407.871,169.795,39.377,157.413
C00735=1039.488,105.724,407.851,169.796,39.377,157.413
C00736=1039.494,105.973,407.831,169.798,39.378,157.413
C00737=1039.501,106.222,407.811,169.800,39.378,157.414
C00738=1039.506,106.472,407.792,169.802,39.378,157.414
C00739=1039.513,106.720,407.772,169.805,39.379,157.414
C00740=1039.519,106.969,407.752,169.807,39.379,157.414
C00741=1039.525,107.219,407.733,169.809,39.379,157.414
C00742=1039.531,107.468,407.713,169.811,39.380,157.414
C00743=1039.537,107.717,407.693,169.813,39.380,157.414
C00744=1039.544,107.966,407.672,169.815,39.381,157.415
C00745=1039.550,108.215,407.654,169.817,39.381,157.415
C00746=1039.556,108.464,407.634,169.820,39.382,157.415
C00747=1039.563,108.750,407.611,169.822,39.382,157.415
C00748=1039.571,109.036,407.588,169.824,39.383,157.415
C00749=1039.578,109.322,407.565,169.827,39.383,157.415
C00750=1039.585,109.608,407.543,169.829,39.384,157.416
C00751=1039.591,109.857,407.523,169.831,39.384,157.416
C00752=1039.598,110.107,407.503,169.834,39.385,157.416
C00753=1039.604,110.355,407.483,169.836,39.385,157.416
C00754=1039.610,110.604,407.463,169.838,39.386,157.416
C00755=1039.616,110.854,407.442,169.840,39.386,157.416
C00756=1039.622,111.103,407.423,169.842,39.387,157.417
C00757=1039.628,111.352,407.403,169.844,39.387,157.417
C00758=1039.635,111.601,407.383,169.846,39.388,157.417
C00759=1039.641,111.850,407.363,169.848,39.388,157.417
C00760=1039.647,112.100,407.343,169.850,39.389,157.417
C00761=1039.653,112.349,407.323,169.852,39.389,157.417
C00762=1039.659,112.597,407.303,169.854,39.390,157.418
C00763=1039.666,112.847,407.282,169.856,39.390,157.418
C00764=1039.672,113.096,407.262,169.858,39.391,157.418
C00765=1039.678,113.345,407.242,169.860,39.391,157.418
C00766=1039.684,113.594,407.222,169.863,39.392,157.418
C00767=1039.690,113.843,407.202,169.865,39.392,157.418
C00768=1039.696,114.092,407.182,169.867,39.393,157.419
C00769=1039.702,114.341,407.161,169.869,39.394,157.419
C00770=1039.708,114.590,407.141,169.871,39.394,157.419
C00771=1039.714,114.839,407.121,169.873,39.395,157.419
C00772=1039.720,115.089,407.100,169.876,39.395,157.419
C00773=1039.726,115.338,407.080,169.878,39.396,157.419
C00774=1039.732,115.587,407.060,169.880,39.396,157.420
C00775=1039.739,115.836,407.040,169.882,39.397,157.420
C00776=1039.744,116.085,407.020,169.883,39.398,157.420
C00777=1039.750,116.335,406.999,169.885,39.398,157.420
C00778=1039.756,116.584,406.979,169.888,39.399,157.420
C00779=1039.763,116.832,406.959,169.890,39.399,157.421
C00780=1039.769,117.082,406.938,169.892,39.400,157.421
C00781=1039.775,117.330,406.918,169.894,39.400,157.421
C00782=1039.781,117.580,406.897,169.896,39.401,157.421
C00783=1039.787,117.829,406.877,169.898,39.401,157.421
C00784=1039.792,118.078,406.857,169.901,39.402,157.421
C00785=1039.799,118.327,406.837,169.903,39.403,157.422
C00786=1039.805,118.576,406.816,169.905,39.403,157.422
C00787=1039.811,118.825,406.795,169.907,39.404,157.422
C00788=1039.817,119.074,406.775,169.909,39.404,157.422
C00789=1039.824,119.324,406.755,169.911,39.405,157.422
C00790=1039.830,119.572,406.735,169.913,39.405,157.422
C00791=1039.835,119.821,406.713,169.916,39.406,157.423
C00792=1039.842,120.071,406.693,169.918,39.406,157.423
C00793=1039.848,120.319,406.673,169.920,39.407,157.423
C00794=1039.854,120.569,406.652,169.922,39.408,157.423
C00795=1039.860,120.817,406.632,169.924,39.408,157.423
C00796=1039.867,121.067,406.611,169.926,39.409,157.424
C00797=1039.872,121.316,406.591,169.929,39.409,157.424
C00798=1039.879,121.565,406.570,169.931,39.410,157.424
C00799=1039.885,121.814,406.550,169.933,39.410,157.424
C00800=1039.891,122.063,406.529,169.935,39.411,157.424
C00801=1039.897,122.312,406.509,169.937,39.411,157.424
C00802=1039.903,122.562,406.488,169.938,39.412,157.425
C00803=1039.910,122.810,406.468,169.941,39.413,157.425
C00804=1039.915,123.060,406.447,169.943,39.413,157.425
C00805=1039.921,123.309,406.427,169.945,39.414,157.425
C00806=1039.928,123.558,406.406,169.947,39.414,157.425
C00807=1039.934,123.807,406.385,169.949,39.415,157.425
C00808=1039.940,124.056,406.365,169.951,39.415,157.426
C00809=1039.946,124.304,406.344,169.953,39.416,157.426
C00810=1039.952,124.554,406.323,169.956,39.416,157.426
C00811=1039.959,124.840,406.300,169.959,39.416,157.426
C00812=1039.967,125.126,406.276,169.961,39.418,157.426
C00813=1039.974,125.412,406.253,169.963,39.418,157.427
C00814=1039.981,125.697,406.229,169.966,39.418,157.427
C00815=1039.988,125.946,406.208,169.968,39.419,157.427
C00816=1039.994,126.196,406.188,169.971,39.419,157.427
C00817=1039.999,126.445,406.167,169.973,39.420,157.427
C00818=1040.006,126.694,406.146,169.975,39.420,157.427
C00819=1040.012,126.942,406.126,169.977,39.421,157.428
C00820=1040.018,127.192,406.105,169.979,39.422,157.428
C00821=1040.025,127.441,406.084,169.981,39.422,157.428
C00822=1040.031,127.689,406.064,169.984,39.423,157.428
C00823=1040.037,127.939,406.043,169.986,39.423,157.428
C00824=1040.043,128.187,406.022,169.988,39.424,157.429
C00825=1040.050,128.437,406.002,169.990,39.424,157.429
C00826=1040.056,128.687,405.981,169.992,39.425,157.429
C00827=1040.062,128.935,405.960,169.994,39.425,157.429
C00828=1040.068,129.185,405.939,169.997,39.426,157.429
C00829=1040.075,129.434,405.918,169.999,39.426,157.429
C00830=1040.081,129.682,405.898,170.001,39.427,157.430
C00831=1040.087,129.932,405.877,170.003,39.427,157.430
C00832=1040.093,130.180,405.856,170.005,39.428,157.430
C00833=1040.100,130.429,405.836,170.007,39.428,157.430
C00834=1040.106,130.678,405.814,170.009,39.429,157.430
C00835=1040.112,130.927,405.794,170.012,39.430,157.430
C00836=1040.118,131.177,405.772,170.014,39.430,157.431
C00837=1040.125,131.426,405.752,170.016,39.431,157.431
C00838=1040.131,131.675,405.731,170.018,39.431,157.431
C00839=1040.137,131.924,405.709,170.020,39.432,157.431
C00840=1040.143,132.173,405.689,170.023,39.433,157.431
C00841=1040.149,132.422,405.667,170.025,39.433,157.432
C00842=1040.156,132.671,405.646,170.027,39.434,157.432
C00843=1040.162,132.920,405.626,170.029,39.434,157.432
C00844=1040.167,133.169,405.604,170.031,39.435,157.432
C00845=1040.174,133.418,405.583,170.034,39.436,157.432
C00846=1040.180,133.667,405.562,170.037,39.436,157.433
C00847=1040.185,133.916,405.541,170.039,39.437,157.433
C00848=1040.192,134.165,405.520,170.041,39.437,157.433
C00849=1040.199,134.414,405.498,170.043,39.438,157.433
C00850=1040.204,134.663,405.477,170.045,39.439,157.433
C00851=1040.211,134.912,405.457,170.047,39.439,157.434
C00852=1040.217,135.162,405.435,170.050,39.440,157.434
C00853=1040.222,135.410,405.414,170.052,39.440,157.434
C00854=1040.229,135.659,405.393,170.054,39.441,157.434
C00855=1040.235,135.909,405.372,170.056,39.442,157.434
C00856=1040.241,136.157,405.351,170.058,39.442,157.434
C00857=1040.248,136.406,405.330,170.060,39.443,157.435
C00858=1040.254,136.655,405.308,170.063,39.443,157.435
C00859=1040.260,136.905,405.286,170.065,39.444,157.435
C00860=1040.266,137.153,405.265,170.067,39.445,157.435
C00861=1040.272,137.403,405.245,170.069,39.445,157.435
C00862=1040.278,137.652,405.223,170.071,39.446,157.436
C00863=1040.284,137.900,405.202,170.074,39.447,157.436
C00864=1040.290,138.149,405.180,170.076,39.447,157.436
C00865=1040.297,138.398,405.159,170.078,39.448,157.436
C00866=1040.303,138.648,405.137,170.081,39.448,157.436
C00867=1040.309,138.896,405.116,170.083,39.449,157.437
C00868=1040.315,139.145,405.095,170.085,39.450,157.437
C00869=1040.322,139.394,405.074,170.088,39.450,157.437
C00870=1040.328,139.644,405.053,170.090,39.451,157.437
C00871=1040.333,139.893,405.031,170.092,39.452,157.437
C00872=1040.339,140.142,405.010,170.094,39.452,157.438
C00873=1040.345,140.391,404.988,170.096,39.453,157.438
C00874=1040.352,140.640,404.966,170.099,39.454,157.438
C00875=1040.358,140.925,404.941,170.101,39.454,157.438
C00876=1040.366,141.211,404.917,170.104,39.455,157.439
C00877=1040.372,141.496,404.892,170.106,39.456,157.439
C00878=1040.380,141.782,404.867,170.108,39.457,157.439
C00879=1040.385,142.031,404.846,170.112,39.457,157.439
C00880=1040.391,142.280,404.824,170.114,39.458,157.439
C00881=1040.397,142.529,404.803,170.116,39.459,157.440
C00882=1040.404,142.778,404.782,170.118,39.459,157.440
C00883=1040.411,143.027,404.760,170.120,39.460,157.440
C00884=1040.416,143.276,404.739,170.123,39.461,157.440
C00885=1040.422,143.525,404.717,170.125,39.461,157.440
C00886=1040.428,143.774,404.695,170.127,39.462,157.441
C00887=1040.435,144.023,404.673,170.129,39.463,157.441
C00888=1040.441,144.272,404.651,170.131,39.463,157.441
C00889=1040.447,144.520,404.630,170.133,39.464,157.441
C00890=1040.453,144.770,404.609,170.136,39.465,157.442
C00891=1040.459,145.019,404.587,170.139,39.465,157.442
C00892=1040.465,145.268,404.565,170.141,39.466,157.442
C00893=1040.471,145.517,404.544,170.143,39.466,157.442
C00894=1040.478,145.766,404.521,170.145,39.467,157.442
C00895=1040.484,146.015,404.500,170.148,39.468,157.442
C00896=1040.489,146.264,404.478,170.150,39.468,157.443
C00897=1040.496,146.513,404.457,170.152,39.470,157.443
C00898=1040.502,146.762,404.435,170.154,39.470,157.443
C00899=1040.508,147.011,404.413,170.156,39.470,157.443
C00900=1040.514,147.260,404.391,170.159,39.472,157.444
C00901=1040.521,147.509,404.369,170.162,39.472,157.444
C00902=1040.527,147.758,404.348,170.164,39.473,157.444
C00903=1040.533,148.007,404.325,170.166,39.474,157.444
C00904=1040.539,148.255,404.304,170.168,39.474,157.444
C00905=1040.545,148.504,404.283,170.171,39.475,157.445
C00906=1040.551,148.753,404.260,170.173,39.476,157.445
C00907=1040.558,149.002,404.239,170.175,39.477,157.445
C00908=1040.563,149.252,404.216,170.177,39.477,157.445
C00909=1040.569,149.500,404.194,170.179,39.478,157.445
C00910=1040.576,149.750,404.172,170.183,39.479,157.446
C00911=1040.582,149.999,404.151,170.185,39.479,157.446
C00912=1040.588,150.247,404.129,170.187,39.480,157.446
C00913=1040.594,150.496,404.107,170.189,39.481,157.446
C00914=1040.599,150.745,404.085,170.192,39.482,157.447
C00915=1040.606,150.994,404.063,170.194,39.482,157.447
C00916=1040.612,151.243,404.041,170.196,39.483,157.447
C00917=1040.618,151.492,404.019,170.198,39.484,157.447
C00918=1040.624,151.741,403.996,170.201,39.484,157.448
C00919=1040.630,151.990,403.974,170.204,39.485,157.448
C00920=1040.636,152.239,403.952,170.206,39.486,157.448
C00921=1040.643,152.488,403.931,170.208,39.487,157.448
C00922=1040.649,152.737,403.908,170.210,39.487,157.448
C00923=1040.654,152.986,403.886,170.212,39.488,157.449
C00924=1040.661,153.235,403.864,170.215,39.489,157.449
C00925=1040.667,153.484,403.842,170.218,39.489,157.449
C00926=1040.674,153.733,403.820,170.220,39.490,157.449
C00927=1040.680,153.982,403.798,170.222,39.491,157.450
C00928=1040.685,154.231,403.775,170.224,39.492,157.450
C00929=1040.692,154.480,403.754,170.227,39.492,157.450
C00930=1040.698,154.729,403.731,170.229,39.494,157.450
C00931=1040.703,154.977,403.709,170.231,39.494,157.450
C00932=1040.709,155.226,403.687,170.234,39.495,157.451
C00933=1040.716,155.475,403.665,170.236,39.496,157.451
C00934=1040.721,155.724,403.642,170.239,39.497,157.451
C00935=1040.728,155.973,403.620,170.241,39.497,157.451
C00936=1040.734,156.221,403.598,170.243,39.498,157.452
C00937=1040.740,156.471,403.575,170.245,39.499,157.452
C00938=1040.746,156.719,403.553,170.249,39.500,157.452
C00939=1040.753,157.005,403.528,170.251,39.500,157.452
C00940=1040.761,157.290,403.502,170.253,39.501,157.453
C00941=1040.767,157.576,403.476,170.256,39.502,157.453
C00942=1040.774,157.861,403.450,170.259,39.503,157.453
C00943=1040.780,158.110,403.428,170.262,39.504,157.453
C00944=1040.787,158.359,403.406,170.264,39.505,157.454
C00945=1040.792,158.608,403.383,170.266,39.505,157.454
C00946=1040.799,158.856,403.361,170.268,39.506,157.454
C00947=1040.804,159.106,403.339,170.271,39.507,157.454
C00948=1040.811,159.354,403.316,170.274,39.508,157.455
C00949=1040.817,159.603,403.294,170.276,39.508,157.455
C00950=1040.823,159.852,403.272,170.278,39.509,157.455
C00951=1040.829,160.101,403.249,170.280,39.510,157.455
C00952=1040.835,160.351,403.226,170.283,39.511,157.456
C00953=1040.842,160.599,403.204,170.285,39.512,157.456
C00954=1040.848,160.848,403.181,170.288,39.513,157.456
C00955=1040.853,161.097,403.158,170.290,39.514,157.456
C00956=1040.859,161.346,403.135,170.293,39.515,157.457
C00957=1040.865,161.595,403.113,170.295,39.516,157.457
C00958=1040.871,161.844,403.090,170.297,39.516,157.457
C00959=1040.877,162.093,403.067,170.299,39.517,157.457
C00960=1040.882,162.342,403.044,170.303,39.518,157.458
C00961=1040.888,162.591,403.021,170.305,39.519,157.458
C00962=1040.895,162.839,402.999,170.307,39.520,157.458
C00963=1040.900,163.088,402.976,170.309,39.521,157.458
C00964=1040.906,163.337,402.953,170.312,39.522,157.459
C00965=1040.912,163.586,402.930,170.314,39.523,157.459
C00966=1040.918,163.835,402.907,170.317,39.524,157.459
C00967=1040.924,164.083,402.885,170.319,39.525,157.460
C00968=1040.930,164.332,402.862,170.322,39.526,157.460
C00969=1040.936,164.581,402.839,170.324,39.527,157.460
C00970=1040.941,164.830,402.816,170.326,39.527,157.460
C00971=1040.947,165.079,402.793,170.329,39.528,157.461
C00972=1040.954,165.328,402.770,170.332,39.529,157.461
C00973=1040.960,165.577,402.747,170.334,39.531,157.461
C00974=1040.966,165.826,402.725,170.336,39.531,157.461
C00975=1040.971,166.075,402.702,170.338,39.532,157.462
C00976=1040.977,166.323,402.678,170.342,39.533,157.462
C00977=1040.984,166.572,402.656,170.344,39.534,157.462
C00978=1040.990,166.821,402.633,170.346,39.535,157.462
C00979=1040.995,167.070,402.610,170.348,39.536,157.463
C00980=1041.002,167.319,402.586,170.351,39.537,157.463
C00981=1041.007,167.568,402.563,170.354,39.538,157.463
C00982=1041.013,167.817,402.540,170.356,39.538,157.464
C00983=1041.020,168.066,402.518,170.358,39.539,157.464
C00984=1041.026,168.314,402.494,170.361,39.541,157.464
C00985=1041.031,168.563,402.472,170.364,39.542,157.464
C00986=1041.038,168.812,402.448,170.366,39.542,157.465
C00987=1041.043,169.061,402.425,170.368,39.543,157.465
C00988=1041.050,169.310,402.403,170.371,39.544,157.465
C00989=1041.056,169.559,402.380,170.374,39.545,157.465
C00990=1041.062,169.807,402.356,170.376,39.546,157.466
C00991=1041.068,170.057,402.333,170.378,39.547,157.466
C00992=1041.074,170.306,402.310,170.381,39.548,157.466
C00993=1041.079,170.554,402.287,170.384,39.549,157.467
C00994=1041.085,170.803,402.263,170.386,39.550,157.467
C00995=1041.092,171.052,402.241,170.388,39.550,157.467
C00996=1041.098,171.301,402.218,170.391,39.552,157.467
C00997=1041.104,171.550,402.195,170.394,39.553,157.468
C00998=1041.110,171.798,402.171,170.396,39.554,157.468
C00999=1041.116,172.048,402.148,170.399,39.554,157.468
C01000=1041.122,172.297,402.125,170.401,39.555,157.468
C01001=1041.129,172.544,402.102,170.404,39.556,157.469
C01002=1041.135,172.793,402.079,170.406,39.557,157.469
C01003=1041.141,173.079,402.052,170.410,39.558,157.469
C01004=1041.149,173.363,402.026,170.412,39.559,157.470
C01005=1041.155,173.648,401.999,170.415,39.560,157.470
C01006=1041.162,173.933,401.972,170.418,39.561,157.470
C01007=1041.169,174.182,401.950,170.421,39.562,157.471
C01008=1041.175,174.431,401.925,170.423,39.564,157.471
C01009=1041.181,174.679,401.903,170.425,39.564,157.471
C01010=1041.187,174.928,401.880,170.429,39.565,157.471
C01011=1041.193,175.177,401.856,170.431,39.566,157.472
C01012=1041.199,175.426,401.833,170.433,39.567,157.472
C01013=1041.205,175.675,401.809,170.436,39.568,157.472
C01014=1041.212,175.924,401.786,170.439,39.569,157.472
C01015=1041.218,176.173,401.763,170.441,39.570,157.473
C01016=1041.224,176.421,401.740,170.444,39.571,157.473
C01017=1041.230,176.671,401.716,170.446,39.572,157.473
C01018=1041.236,176.919,401.693,170.449,39.573,157.474
C01019=1041.243,177.168,401.669,170.452,39.573,157.474
C01020=1041.249,177.417,401.646,170.454,39.574,157.474
C01021=1041.255,177.666,401.623,170.456,39.575,157.474
C01022=1041.261,177.915,401.599,170.460,39.576,157.475
C01023=1041.267,178.164,401.576,170.462,39.578,157.475
C01024=1041.274,178.412,401.552,170.464,39.578,157.475
C01025=1041.280,178.660,401.529,170.467,39.579,157.476
C01026=1041.286,178.909,401.506,170.470,39.580,157.476
C01027=1041.293,179.158,401.482,170.472,39.581,157.476
C01028=1041.298,179.407,401.459,170.475,39.582,157.476
C01029=1041.305,179.656,401.435,170.478,39.583,157.477
C01030=1041.311,179.905,401.412,170.481,39.584,157.477
C01031=1041.317,180.154,401.388,170.483,39.585,157.477
C01032=1041.323,180.402,401.364,170.485,39.586,157.477
C01033=1041.330,180.652,401.341,170.489,39.587,157.478
C01034=1041.337,180.900,401.318,170.491,39.588,157.478
C01035=1041.343,181.149,401.294,170.493,39.589,157.478
C01036=1041.349,181.398,401.271,170.496,39.589,157.479
C01037=1041.356,181.647,401.247,170.499,39.590,157.479
C01038=1041.362,181.895,401.223,170.502,39.591,157.479
C01039=1041.368,182.145,401.200,170.504,39.593,157.480
C01040=1041.374,182.393,401.176,170.507,39.594,157.480
C01041=1041.381,182.642,401.152,170.510,39.595,157.480
C01042=1041.386,182.891,401.129,170.512,39.596,157.480
C01043=1041.393,183.140,401.105,170.515,39.596,157.481
C01044=1041.399,183.388,401.081,170.518,39.597,157.481
C01045=1041.406,183.637,401.057,170.520,39.598,157.481
C01046=1041.411,183.886,401.034,170.523,39.599,157.482
C01047=1041.417,184.135,401.010,170.525,39.600,157.482
C01048=1041.423,184.384,400.986,170.529,39.602,157.482
C01049=1041.429,184.632,400.962,170.531,39.603,157.483
C01050=1041.435,184.881,400.938,170.533,39.604,157.483
C01051=1041.441,185.130,400.914,170.537,39.605,157.483
C01052=1041.447,185.379,400.890,170.539,39.606,157.483
C01053=1041.453,185.627,400.865,170.541,39.607,157.484
C01054=1041.459,185.876,400.841,170.545,39.609,157.484
C01055=1041.465,186.124,400.818,170.547,39.610,157.485
C01056=1041.471,186.374,400.793,170.549,39.611,157.485
C01057=1041.477,186.622,400.769,170.553,39.612,157.485
C01058=1041.483,186.871,400.745,170.555,39.613,157.485
C01059=1041.489,187.120,400.721,170.558,39.615,157.486
C01060=1041.495,187.369,400.696,170.561,39.616,157.486
C01061=1041.501,187.617,400.673,170.563,39.617,157.486
C01062=1041.507,187.866,400.648,170.566,39.618,157.487
C01063=1041.513,188.115,400.625,170.568,39.619,157.487
C01064=1041.519,188.364,400.600,170.572,39.621,157.488
C01065=1041.525,188.612,400.576,170.574,39.622,157.488
C01066=1041.531,188.861,400.551,170.576,39.623,157.488
C01067=1041.538,189.146,400.524,170.580,39.624,157.488
C01068=1041.545,189.429,400.496,170.583,39.625,157.489
C01069=1041.552,189.714,400.468,170.587,39.627,157.489
C01070=1041.559,189.999,400.440,170.589,39.628,157.490
C01071=1041.565,190.247,400.416,170.592,39.629,157.490
C01072=1041.571,190.496,400.392,170.595,39.631,157.490
C01073=1041.577,190.745,400.368,170.598,39.632,157.491
C01074=1041.582,190.994,400.343,170.600,39.633,157.491
C01075=1041.589,191.243,400.319,170.604,39.634,157.491
C01076=1041.595,191.491,400.294,170.606,39.635,157.492
C01077=1041.601,191.740,400.270,170.608,39.637,157.492
C01078=1041.607,191.989,400.246,170.612,39.638,157.492
C01079=1041.613,192.237,400.222,170.614,39.639,157.493
C01080=1041.619,192.486,400.197,170.617,39.640,157.493
C01081=1041.626,192.734,400.173,170.620,39.641,157.493
C01082=1041.631,192.984,400.148,170.623,39.642,157.494
C01083=1041.638,193.233,400.124,170.625,39.644,157.494
C01084=1041.644,193.481,400.099,170.628,39.645,157.494
C01085=1041.650,193.730,400.075,170.631,39.646,157.495
C01086=1041.656,193.979,400.051,170.634,39.647,157.495
C01087=1041.662,194.227,400.026,170.636,39.648,157.495
C01088=1041.668,194.476,400.002,170.640,39.650,157.496
C01089=1041.674,194.725,399.977,170.642,39.651,157.496
C01090=1041.681,194.973,399.952,170.645,39.652,157.497
C01091=1041.687,195.222,399.928,170.648,39.653,157.497
C01092=1041.693,195.471,399.904,170.651,39.655,157.497
C01093=1041.699,195.720,399.879,170.653,39.656,157.498
C01094=1041.705,195.968,399.855,170.657,39.657,157.498
C01095=1041.712,196.217,399.830,170.659,39.658,157.498
C01096=1041.718,196.466,399.805,170.662,39.659,157.499
C01097=1041.724,196.715,399.781,170.665,39.660,157.499
C01098=1041.730,196.963,399.756,170.668,39.661,157.499
C01099=1041.736,197.212,399.732,170.670,39.663,157.500
C01100=1041.743,197.460,399.707,170.674,39.664,157.500
C01101=1041.749,197.709,399.683,170.676,39.665,157.500
C01102=1041.755,197.957,399.658,170.680,39.667,157.501
C01103=1041.761,198.207,399.633,170.682,39.668,157.501
C01104=1041.768,198.455,399.608,170.685,39.669,157.501
C01105=1041.774,198.704,399.584,170.688,39.671,157.502
C01106=1041.781,198.953,399.559,170.691,39.672,157.502
C01107=1041.786,199.201,399.535,170.693,39.673,157.502
C01108=1041.793,199.450,399.510,170.697,39.674,157.503
C01109=1041.799,199.699,399.485,170.699,39.675,157.503
C01110=1041.805,199.948,399.460,170.702,39.676,157.503
C01111=1041.812,200.196,399.435,170.706,39.678,157.504
C01112=1041.818,200.445,399.411,170.708,39.679,157.504
C01113=1041.825,200.694,399.386,170.711,39.680,157.505
C01114=1041.830,200.942,399.362,170.714,39.682,157.505
C01115=1041.836,201.191,399.336,170.717,39.683,157.505
C01116=1041.842,201.440,399.311,170.719,39.684,157.506
C01117=1041.848,201.689,399.286,170.723,39.685,157.506
C01118=1041.855,201.937,399.262,170.725,39.687,157.507
C01119=1041.861,202.186,399.236,170.728,39.688,157.507
C01120=1041.867,202.434,399.211,170.732,39.690,157.507
C01121=1041.873,202.682,399.186,170.734,39.691,157.508
C01122=1041.879,202.932,399.161,170.738,39.692,157.508
C01123=1041.885,203.180,399.136,170.740,39.694,157.508
C01124=1041.892,203.429,399.111,170.743,39.695,157.509
C01125=1041.898,203.678,399.085,170.746,39.697,157.509
C01126=1041.904,203.926,399.060,170.749,39.698,157.510
C01127=1041.909,204.175,399.036,170.751,39.699,157.510
C01128=1041.916,204.424,399.010,170.755,39.701,157.510
C01129=1041.922,204.672,398.985,170.758,39.702,157.511
C01130=1041.928,204.921,398.960,170.761,39.704,157.511
C01131=1041.954,205.972,398.853,171.038,39.806,157.543
C01132=1041.962,206.268,398.822,171.040,39.808,157.543
C01133=1041.970,206.564,398.791,171.043,39.811,157.544
C01134=1041.979,206.860,398.759,171.045,39.814,157.544
C01135=1041.987,207.156,398.728,171.048,39.817,157.545
C01136=1041.992,207.405,398.702,171.051,39.818,157.546
C01137=1042.000,207.653,398.675,171.052,39.821,157.546
C01138=1042.006,207.901,398.649,171.055,39.823,157.547
C01139=1042.013,208.150,398.623,171.057,39.825,157.547
C01140=1042.019,208.399,398.596,171.059,39.827,157.548
C01141=1042.026,208.647,398.570,171.061,39.829,157.548
C01142=1042.033,208.896,398.543,171.064,39.831,157.549
C01143=1042.039,209.144,398.517,171.065,39.833,157.549
C01144=1042.046,209.393,398.490,171.068,39.836,157.550
C01145=1042.053,209.641,398.463,171.071,39.838,157.550
C01146=1042.059,209.890,398.436,171.072,39.840,157.551
C01147=1042.066,210.138,398.410,171.075,39.842,157.551
C01148=1042.073,210.386,398.384,171.077,39.844,157.552
C01149=1042.079,210.636,398.357,171.079,39.847,157.553
C01150=1042.086,210.884,398.331,171.081,39.848,157.553
C01151=1042.092,211.133,398.304,171.084,39.850,157.554
C01152=1042.099,211.381,398.278,171.085,39.853,157.554
C01153=1042.106,211.629,398.251,171.088,39.855,157.555
C01154=1042.112,211.878,398.224,171.090,39.857,157.555
C01155=1042.119,212.126,398.198,171.092,39.859,157.556
C01156=1042.125,212.375,398.171,171.095,39.861,157.556
C01157=1042.131,212.623,398.143,171.097,39.863,157.557
C01158=1042.139,212.872,398.117,171.099,39.866,157.557
C01159=1042.145,213.121,398.090,171.101,39.868,157.558
C01160=1042.151,213.369,398.064,171.104,39.870,157.558
C01161=1042.158,213.617,398.036,171.105,39.872,157.559
C01162=1042.165,213.866,398.010,171.108,39.874,157.559
C01163=1042.171,214.114,397.983,171.110,39.876,157.560
C01164=1042.178,214.362,397.956,171.112,39.879,157.561
C01165=1042.184,214.611,397.929,171.114,39.880,157.561
C01166=1042.191,214.860,397.902,171.117,39.883,157.562
C01167=1042.198,215.108,397.875,171.120,39.885,157.562
C01168=1042.204,215.356,397.848,171.121,39.887,157.563
C01169=1042.211,215.605,397.822,171.124,39.889,157.563
C01170=1042.218,215.853,397.794,171.126,39.891,157.564
C01171=1042.224,216.101,397.768,171.128,39.894,157.564
C01172=1042.230,216.351,397.741,171.130,39.895,157.565
C01173=1042.237,216.599,397.713,171.133,39.898,157.565
C01174=1042.244,216.848,397.687,171.135,39.900,157.566
C01175=1042.250,217.095,397.660,171.137,39.902,157.566
C01176=1042.257,217.344,397.633,171.139,39.904,157.567
C01177=1042.264,217.593,397.606,171.142,39.906,157.567
C01178=1042.271,217.841,397.579,171.144,39.908,157.568
C01179=1042.277,218.090,397.552,171.146,39.910,157.568
C01180=1042.284,218.338,397.525,171.149,39.913,157.569
C01181=1042.291,218.587,397.498,171.151,39.914,157.569
C01182=1042.297,218.835,397.471,171.154,39.916,157.570
C01183=1042.304,219.083,397.444,171.155,39.919,157.571
C01184=1042.311,219.332,397.417,171.158,39.920,157.571
C01185=1042.317,219.581,397.390,171.160,39.923,157.572
C01186=1042.324,219.828,397.363,171.163,39.925,157.572
C01187=1042.330,220.077,397.336,171.165,39.927,157.573
C01188=1042.339,220.379,397.303,171.168,39.930,157.573
C01189=1042.346,220.680,397.270,171.171,39.932,157.574
C01190=1042.354,220.982,397.236,171.173,39.935,157.575
C01191=1042.362,221.283,397.203,171.176,39.938,157.575
C01192=1042.369,221.532,397.176,171.179,39.939,157.576
C01193=1042.376,221.780,397.149,171.181,39.942,157.576
C01194=1042.382,222.028,397.122,171.183,39.944,157.577
C01195=1042.389,222.277,397.094,171.185,39.946,157.578
C01196=1042.395,222.526,397.067,171.188,39.948,157.578
C01197=1042.402,222.774,397.039,171.190,39.950,157.579
C01198=1042.408,223.022,397.012,171.193,39.952,157.579
C01199=1042.414,223.271,396.985,171.194,39.955,157.580
C01200=1042.422,223.519,396.958,171.197,39.956,157.580
C01201=1042.428,223.768,396.930,171.200,39.959,157.581
C01202=1042.435,224.016,396.902,171.202,39.961,157.581
C01203=1042.441,224.264,396.876,171.205,39.963,157.582
C01204=1042.447,224.513,396.848,171.206,39.965,157.582
C01205=1042.454,224.761,396.820,171.209,39.967,157.583
C01206=1042.461,225.010,396.793,171.211,39.970,157.583
C01207=1042.468,225.258,396.765,171.214,39.971,157.584
C01208=1042.475,225.507,396.738,171.216,39.973,157.584
C01209=1042.481,225.755,396.711,171.219,39.976,157.585
C01210=1042.487,226.003,396.683,171.222,39.978,157.586
C01211=1042.494,226.251,396.656,171.223,39.980,157.586
C01212=1042.501,226.500,396.628,171.226,39.982,157.587
C01213=1042.507,226.749,396.601,171.228,39.984,157.587
C01214=1042.514,226.997,396.573,171.231,39.986,157.588
C01215=1042.521,227.246,396.546,171.233,39.988,157.588
C01216=1042.528,227.494,396.518,171.236,39.990,157.589
C01217=1042.535,227.742,396.491,171.238,39.992,157.589
C01218=1042.541,227.990,396.463,171.240,39.994,157.590
C01219=1042.547,228.239,396.435,171.243,39.997,157.590
C01220=1042.554,228.487,396.408,171.245,39.999,157.591
C01221=1042.561,228.735,396.380,171.248,40.001,157.591
C01222=1042.567,228.984,396.352,171.250,40.003,157.592
C01223=1042.574,229.232,396.325,171.253,40.005,157.593
C01224=1042.581,229.481,396.297,171.255,40.007,157.593
C01225=1042.587,229.729,396.269,171.258,40.009,157.594
C01226=1042.594,229.978,396.241,171.259,40.011,157.594
C01227=1042.600,230.226,396.213,171.262,40.014,157.595
C01228=1042.606,230.474,396.186,171.265,40.016,157.595
C01229=1042.613,230.723,396.158,171.267,40.018,157.596
C01230=1042.619,230.971,396.130,171.270,40.020,157.596
C01231=1042.626,231.219,396.102,171.272,40.022,157.597
C01232=1042.633,231.468,396.075,171.275,40.024,157.598
C01233=1042.640,231.716,396.047,171.277,40.026,157.598
C01234=1042.646,231.965,396.019,171.280,40.028,157.599
C01235=1042.652,232.213,395.990,171.282,40.031,157.599
C01236=1042.659,232.461,395.963,171.284,40.033,157.600
C01237=1042.666,232.710,395.935,171.287,40.035,157.600
C01238=1042.673,232.958,395.907,171.289,40.037,157.601
C01239=1042.678,233.207,395.879,171.292,40.039,157.601
C01240=1042.685,233.455,395.850,171.294,40.041,157.602
C01241=1042.692,233.703,395.823,171.297,40.044,157.603
C01242=1042.699,233.952,395.795,171.300,40.046,157.603
C01243=1042.705,234.200,395.766,171.302,40.048,157.604
C01244=1042.713,234.494,395.734,171.305,40.050,157.604
C01245=1042.721,234.788,395.700,171.307,40.053,157.605
C01246=1042.728,235.082,395.667,171.311,40.055,157.606
C01247=1042.736,235.376,395.634,171.314,40.058,157.606
C01248=1042.743,235.624,395.606,171.316,40.060,157.607
C01249=1042.749,235.872,395.577,171.319,40.062,157.607
C01250=1042.756,236.121,395.549,171.322,40.064,157.608
C01251=1042.762,236.369,395.522,171.324,40.066,157.608
C01252=1042.769,236.617,395.493,171.327,40.068,157.609
C01253=1042.775,236.866,395.465,171.329,40.071,157.610
C01254=1042.782,237.114,395.437,171.332,40.073,157.610
C01255=1042.789,237.362,395.409,171.334,40.075,157.611
C01256=1042.795,237.611,395.380,171.337,40.077,157.611
C01257=1042.802,237.860,395.352,171.340,40.079,157.612
C01258=1042.809,238.108,395.324,171.342,40.081,157.612
C01259=1042.816,238.356,395.296,171.345,40.084,157.613
C01260=1042.822,238.605,395.267,171.347,40.085,157.613
C01261=1042.829,238.853,395.239,171.350,40.087,157.614
C01262=1042.835,239.101,395.210,171.352,40.090,157.615
C01263=1042.842,239.350,395.182,171.355,40.092,157.615
C01264=1042.849,239.597,395.154,171.358,40.094,157.616
C01265=1042.855,239.846,395.126,171.360,40.096,157.616
C01266=1042.862,240.094,395.097,171.363,40.098,157.617
C01267=1042.868,240.342,395.069,171.365,40.100,157.617
C01268=1042.875,240.591,395.040,171.368,40.103,157.618
C01269=1042.882,240.840,395.012,171.370,40.104,157.618
C01270=1042.889,241.087,394.984,171.373,40.106,157.619
C01271=1042.895,241.336,394.956,171.376,40.109,157.620
C01272=1042.902,241.584,394.927,171.378,40.111,157.620
C01273=1042.908,241.832,394.898,171.381,40.113,157.621
C01274=1042.914,242.081,394.870,171.383,40.115,157.621
C01275=1042.921,242.329,394.841,171.386,40.118,157.622
C01276=1042.927,242.577,394.812,171.388,40.119,157.622
C01277=1042.934,242.826,394.784,171.391,40.122,157.623
C01278=1042.941,243.074,394.755,171.394,40.124,157.623
C01279=1042.947,243.322,394.726,171.396,40.126,157.624
C01280=1042.954,243.571,394.698,171.399,40.128,157.625
C01281=1042.960,243.819,394.669,171.402,40.131,157.625
C01282=1042.967,244.067,394.641,171.404,40.133,157.626
C01283=1042.973,244.315,394.612,171.407,40.134,157.626
C01284=1042.980,244.564,394.583,171.409,40.137,157.627
C01285=1042.987,244.812,394.555,171.412,40.139,157.627
C01286=1042.993,245.060,394.526,171.414,40.141,157.628
C01287=1043.000,245.308,394.497,171.417,40.143,157.629
C01288=1043.006,245.557,394.469,171.420,40.146,157.629
C01289=1043.012,245.805,394.440,171.422,40.148,157.630
C01290=1043.019,246.054,394.410,171.426,40.150,157.630
C01291=1043.025,246.302,394.381,171.429,40.152,157.631
C01292=1043.031,246.550,394.352,171.431,40.155,157.632
C01293=1043.038,246.798,394.323,171.434,40.157,157.632
C01294=1043.045,247.046,394.295,171.436,40.159,157.633
C01295=1043.051,247.294,394.266,171.439,40.161,157.633
C01296=1043.058,247.543,394.236,171.442,40.164,157.634
C01297=1043.064,247.791,394.207,171.444,40.165,157.634
C01298=1043.070,248.039,394.178,171.447,40.167,157.635
C01299=1043.076,248.287,394.149,171.449,40.170,157.636
C01300=1043.084,248.576,394.116,171.453,40.172,157.636
C01301=1043.091,248.864,394.082,171.456,40.175,157.637
C01302=1043.099,249.152,394.048,171.458,40.178,157.638
C01303=1043.106,249.440,394.015,171.462,40.180,157.638
C01304=1043.113,249.688,393.986,171.465,40.183,157.639
C01305=1043.120,249.937,393.957,171.467,40.185,157.640
C01306=1043.126,250.185,393.928,171.470,40.187,157.640
C01307=1043.133,250.433,393.899,171.473,40.189,157.641
C01308=1043.139,250.681,393.869,171.475,40.191,157.641
C01309=1043.146,250.930,393.840,171.479,40.193,157.642
C01310=1043.152,251.178,393.811,171.481,40.195,157.642
C01311=1043.159,251.426,393.782,171.484,40.197,157.643
C01312=1043.166,251.675,393.752,171.487,40.200,157.644
C01313=1043.172,251.923,393.724,171.489,40.202,157.644
C01314=1043.179,252.171,393.695,171.492,40.204,157.645
C01315=1043.185,252.419,393.666,171.494,40.206,157.645
C01316=1043.192,252.667,393.635,171.498,40.209,157.646
C01317=1043.198,252.915,393.606,171.501,40.211,157.647
C01318=1043.205,253.163,393.577,171.503,40.213,157.647
C01319=1043.211,253.412,393.548,171.506,40.215,157.648
C01320=1043.218,253.660,393.518,171.509,40.218,157.648
C01321=1043.225,253.908,393.489,171.511,40.220,157.649
C01322=1043.231,254.157,393.460,171.515,40.222,157.650
C01323=1043.237,254.405,393.431,171.517,40.224,157.650
C01324=1043.245,254.653,393.401,171.520,40.226,157.651
C01325=1043.252,254.901,393.372,171.523,40.228,157.651
C01326=1043.258,255.149,393.343,171.525,40.230,157.652
C01327=1043.265,255.398,393.314,171.529,40.232,157.652
C01328=1043.271,255.645,393.284,171.531,40.235,157.653
C01329=1043.278,255.894,393.255,171.534,40.237,157.654
C01330=1043.284,256.142,393.226,171.537,40.239,157.654
C01331=1043.291,256.390,393.196,171.539,40.241,157.655
C01332=1043.298,256.639,393.166,171.543,40.243,157.655
C01333=1043.304,256.886,393.137,171.546,40.246,157.656
C01334=1043.311,257.135,393.107,171.548,40.248,157.657
C01335=1043.317,257.383,393.078,171.551,40.250,157.657
C01336=1043.325,257.631,393.048,171.554,40.252,157.658
C01337=1043.332,257.879,393.020,171.557,40.254,157.658
C01338=1043.339,258.127,392.989,171.560,40.257,157.659
C01339=1043.345,258.375,392.960,171.562,40.259,157.660
C01340=1043.352,258.624,392.931,171.566,40.260,157.660
C01341=1043.358,258.872,392.901,171.568,40.263,157.661
C01342=1043.365,259.121,392.872,171.571,40.265,157.661
C01343=1043.372,259.368,392.842,171.574,40.267,157.662
C01344=1043.379,259.617,392.813,171.577,40.269,157.662
C01345=1043.385,259.864,392.783,171.580,40.271,157.663
C01346=1043.392,260.113,392.754,171.583,40.274,157.664
C01347=1043.399,260.361,392.724,171.586,40.276,157.664
C01348=1043.406,260.609,392.694,171.589,40.278,157.665
C01349=1043.412,260.857,392.665,171.591,40.280,157.665
C01350=1043.419,261.105,392.634,171.594,40.282,157.666
C01351=1043.425,261.353,392.605,171.598,40.285,157.667
C01352=1043.433,261.602,392.575,171.600,40.287,157.667
C01353=1043.439,261.850,392.546,171.603,40.289,157.668
C01354=1043.446,262.098,392.516,171.606,40.291,157.668
C01355=1043.453,262.346,392.486,171.609,40.293,157.669
C01356=1043.461,262.633,392.452,171.613,40.296,157.670
C01357=1043.468,262.919,392.417,171.616,40.298,157.670
C01358=1043.476,263.207,392.383,171.619,40.301,157.671
C01359=1043.483,263.493,392.348,171.622,40.303,157.672
C01360=1043.490,263.741,392.318,171.626,40.306,157.672
C01361=1043.496,263.989,392.288,171.628,40.308,157.673
C01362=1043.503,264.238,392.258,171.631,40.310,157.674
C01363=1043.510,264.485,392.228,171.635,40.313,157.674
C01364=1043.516,264.734,392.197,171.637,40.315,157.675
C01365=1043.522,264.982,392.168,171.640,40.317,157.675
C01366=1043.530,265.230,392.138,171.644,40.319,157.676
C01367=1043.535,265.478,392.108,171.646,40.321,157.677
C01368=1043.543,265.726,392.078,171.649,40.324,157.677
C01369=1043.550,265.974,392.047,171.653,40.326,157.678
C01370=1043.556,266.222,392.017,171.655,40.329,157.679
C01371=1043.563,266.470,391.987,171.658,40.331,157.679
C01372=1043.569,266.718,391.957,171.662,40.333,157.680
C01373=1043.576,266.966,391.926,171.664,40.335,157.680
C01374=1043.583,267.215,391.896,171.667,40.337,157.681
C01375=1043.589,267.462,391.867,171.670,40.339,157.682
C01376=1043.596,267.711,391.836,171.673,40.342,157.682
C01377=1043.603,267.959,391.806,171.676,40.344,157.683
C01378=1043.609,268.207,391.775,171.680,40.347,157.684
C01379=1043.616,268.455,391.745,171.682,40.349,157.684
C01380=1043.622,268.703,391.715,171.685,40.351,157.685
C01381=1043.629,268.951,391.685,171.688,40.353,157.685
C01382=1043.635,269.199,391.654,171.691,40.355,157.686
C01383=1043.642,269.447,391.624,171.695,40.358,157.687
C01384=1043.648,269.695,391.594,171.698,40.360,157.687
C01385=1043.655,269.944,391.563,171.700,40.362,157.688
C01386=1043.662,270.191,391.532,171.704,40.365,157.689
C01387=1043.669,270.439,391.502,171.706,40.367,157.689
C01388=1043.675,270.688,391.472,171.709,40.369,157.690
C01389=1043.682,270.936,391.441,171.713,40.372,157.690
C01390=1043.688,271.184,391.411,171.715,40.374,157.691
C01391=1043.696,271.431,391.380,171.719,40.376,157.692
C01392=1043.702,271.680,391.350,171.722,40.378,157.692
C01393=1043.709,271.927,391.320,171.725,40.381,157.693
C01394=1043.715,272.176,391.289,171.728,40.383,157.694
C01395=1043.722,272.424,391.258,171.731,40.385,157.694
C01396=1043.729,272.672,391.228,171.734,40.387,157.695
C01397=1043.735,272.920,391.197,171.737,40.390,157.696
C01398=1043.741,273.168,391.166,171.741,40.392,157.696
C01399=1043.749,273.416,391.136,171.744,40.395,157.697
C01400=1043.754,273.664,391.105,171.746,40.397,157.697
C01401=1043.761,273.912,391.074,171.750,40.400,157.698
C01402=1043.768,274.160,391.044,171.753,40.402,157.699
C01403=1043.775,274.408,391.012,171.756,40.404,157.699
C01404=1043.781,274.655,390.982,171.759,40.406,157.700
C01405=1043.788,274.904,390.952,171.763,40.409,157.701
C01406=1043.795,275.152,390.920,171.765,40.411,157.701
C01407=1043.801,275.400,390.890,171.768,40.413,157.702
C01408=1043.808,275.648,390.858,171.772,40.416,157.703
C01409=1043.814,275.896,390.828,171.774,40.418,157.703
C01410=1043.821,276.143,390.797,171.778,40.420,157.704
C01411=1043.828,276.392,390.766,171.781,40.423,157.705
C01412=1043.835,276.683,390.730,171.785,40.426,157.705
C01413=1043.844,276.974,390.693,171.788,40.428,157.706
C01414=1043.851,277.266,390.657,171.792,40.431,157.707
C01415=1043.859,277.556,390.621,171.796,40.434,157.708
C01416=1043.866,277.804,390.589,171.799,40.436,157.708
C01417=1043.873,278.053,390.559,171.803,40.439,157.709
C01418=1043.880,278.300,390.528,171.805,40.441,157.710
C01419=1043.886,278.549,390.497,171.809,40.443,157.710
C01420=1043.892,278.796,390.466,171.812,40.446,157.711
C01421=1043.899,279.044,390.435,171.815,40.448,157.712
C01422=1043.905,279.293,390.404,171.818,40.450,157.712
C01423=1043.912,279.541,390.373,171.822,40.453,157.713
C01424=1043.919,279.788,390.341,171.824,40.455,157.714
C01425=1043.925,280.036,390.310,171.828,40.458,157.714
C01426=1043.932,280.284,390.278,171.831,40.460,157.715
C01427=1043.938,280.532,390.248,171.835,40.463,157.716
C01428=1043.945,280.780,390.216,171.837,40.465,157.716
C01429=1043.951,281.028,390.185,171.841,40.467,157.717
C01430=1043.958,281.276,390.154,171.845,40.470,157.718
C01431=1043.965,281.524,390.122,171.848,40.472,157.719
C01432=1043.972,281.772,390.091,171.851,40.474,157.719
C01433=1043.978,282.020,390.060,171.854,40.477,157.720
C01434=1043.985,282.268,390.029,171.858,40.479,157.721
C01435=1043.991,282.516,389.997,171.860,40.482,157.721
C01436=1043.998,282.764,389.966,171.864,40.484,157.722
C01437=1044.005,283.012,389.934,171.867,40.486,157.722
C01438=1044.012,283.260,389.903,171.871,40.489,157.723
C01439=1044.018,283.508,389.871,171.873,40.491,157.724
C01440=1044.025,283.755,389.840,171.877,40.494,157.725
C01441=1044.032,284.003,389.809,171.881,40.496,157.725
C01442=1044.038,284.251,389.777,171.883,40.499,157.726
C01443=1044.045,284.499,389.746,171.887,40.501,157.727
C01444=1044.052,284.747,389.714,171.890,40.504,157.727
C01445=1044.059,284.995,389.683,171.894,40.506,157.728
C01446=1044.065,285.243,389.651,171.897,40.508,157.729
C01447=1044.072,285.491,389.620,171.900,40.511,157.729
C01448=1044.079,285.739,389.588,171.904,40.513,157.730
C01449=1044.086,285.987,389.557,171.907,40.516,157.731
C01450=1044.092,286.234,389.526,171.910,40.518,157.731
C01451=1044.099,286.482,389.493,171.914,40.520,157.732
C01452=1044.106,286.730,389.462,171.917,40.523,157.733
C01453=1044.113,286.978,389.431,171.920,40.525,157.733
C01454=1044.120,287.225,389.399,171.923,40.528,157.734
C01455=1044.125,287.474,389.367,171.927,40.531,157.735
C01456=1044.132,287.722,389.336,171.931,40.533,157.736
C01457=1044.139,287.969,389.304,171.934,40.536,157.736
C01458=1044.146,288.217,389.272,171.937,40.538,157.737
C01459=1044.153,288.465,389.241,171.941,40.540,157.738
C01460=1044.159,288.712,389.208,171.944,40.543,157.739
C01461=1044.166,288.960,389.177,171.948,40.545,157.739
C01462=1044.173,289.209,389.145,171.950,40.548,157.740
C01463=1044.180,289.456,389.113,171.954,40.551,157.741
C01464=1044.186,289.704,389.081,171.958,40.553,157.741
C01465=1044.193,289.952,389.049,171.961,40.555,157.742
C01466=1044.200,290.199,389.017,171.964,40.558,157.743
C01467=1044.206,290.448,388.985,171.968,40.560,157.743
C01468=1044.215,290.751,388.947,171.972,40.564,157.744
C01469=1044.223,291.053,388.907,171.976,40.567,157.745
C01470=1044.231,291.357,388.868,171.981,40.569,157.746
C01471=1044.239,291.659,388.828,171.985,40.573,157.747
C01472=1044.246,291.907,388.797,171.988,40.575,157.748
C01473=1044.252,292.155,388.764,171.992,40.578,157.748
C01474=1044.259,292.403,388.733,171.995,40.580,157.749
C01475=1044.266,292.650,388.701,171.999,40.583,157.750
C01476=1044.273,292.899,388.668,172.002,40.586,157.751
C01477=1044.280,293.146,388.636,172.006,40.588,157.751
C01478=1044.287,293.394,388.604,172.009,40.590,157.752
C01479=1044.293,293.642,388.572,172.012,40.593,157.753
C01480=1044.300,293.889,388.540,172.016,40.596,157.754
C01481=1044.306,294.138,388.507,172.020,40.598,157.754
C01482=1044.313,294.385,388.475,172.023,40.601,157.755
C01483=1044.320,294.633,388.442,172.026,40.603,157.756
C01484=1044.326,294.881,388.411,172.030,40.606,157.756
C01485=1044.333,295.128,388.378,172.034,40.609,157.757
C01486=1044.340,295.376,388.346,172.037,40.611,157.758
C01487=1044.347,295.624,388.313,172.040,40.613,157.759
C01488=1044.353,295.872,388.282,172.044,40.616,157.759
C01489=1044.360,296.119,388.249,172.048,40.619,157.760
C01490=1044.367,296.368,388.216,172.051,40.622,157.761
C01491=1044.373,296.615,388.183,172.055,40.624,157.762
C01492=1044.380,296.863,388.151,172.059,40.627,157.762
C01493=1044.386,297.110,388.118,172.062,40.630,157.763
C01494=1044.392,297.358,388.085,172.065,40.632,157.764
C01495=1044.399,297.606,388.052,172.069,40.635,157.765
C01496=1044.406,297.853,388.020,172.073,40.638,157.766
C01497=1044.413,298.101,387.987,172.076,40.640,157.766
C01498=1044.420,298.349,387.954,172.080,40.643,157.767
C01499=1044.426,298.597,387.921,172.083,40.646,157.768
C01500=1044.432,298.844,387.889,172.087,40.648,157.769
C01501=1044.439,299.092,387.857,172.091,40.651,157.769
C01502=1044.446,299.340,387.823,172.094,40.654,157.770
C01503=1044.452,299.588,387.791,172.098,40.656,157.771
C01504=1044.459,299.835,387.758,172.101,40.659,157.772
C01505=1044.466,300.083,387.725,172.105,40.662,157.772
C01506=1044.473,300.331,387.693,172.108,40.665,157.773
C01507=1044.479,300.578,387.660,172.112,40.667,157.774
C01508=1044.486,300.827,387.627,172.116,40.670,157.775
C01509=1044.492,301.074,387.594,172.120,40.673,157.776
C01510=1044.498,301.322,387.561,172.123,40.675,157.776
C01511=1044.506,301.569,387.528,172.126,40.679,157.777
C01512=1044.513,301.817,387.495,172.130,40.681,157.778
C01513=1044.519,302.065,387.462,172.134,40.684,157.779
C01514=1044.526,302.313,387.430,172.138,40.687,157.780
C01515=1044.532,302.560,387.397,172.142,40.689,157.780
C01516=1044.539,302.808,387.363,172.146,40.692,157.781
C01517=1044.546,303.055,387.331,172.148,40.695,157.782
C01518=1044.553,303.304,387.298,172.152,40.697,157.783
C01519=1044.560,303.550,387.264,172.156,40.700,157.783
C01520=1044.567,303.799,387.231,172.160,40.703,157.784
C01521=1044.573,304.046,387.198,172.164,40.705,157.785
C01522=1044.580,304.293,387.165,172.168,40.708,157.786
C01523=1044.587,304.541,387.132,172.172,40.711,157.787
C01524=1044.596,304.861,387.090,172.176,40.714,157.788
C01525=1044.604,305.180,387.047,172.181,40.718,157.789
C01526=1044.613,305.499,387.004,172.186,40.722,157.790
C01527=1044.623,305.818,386.961,172.191,40.725,157.791
C01528=1044.629,306.066,386.928,172.194,40.728,157.791
C01529=1044.636,306.314,386.895,172.198,40.731,157.792
C01530=1044.642,306.561,386.862,172.202,40.733,157.793
C01531=1044.649,306.810,386.829,172.206,40.736,157.794
C01532=1044.656,307.057,386.795,172.209,40.739,157.795
C01533=1044.663,307.305,386.763,172.213,40.741,157.795
C01534=1044.671,307.552,386.729,172.217,40.744,157.796
C01535=1044.677,307.799,386.696,172.221,40.747,157.797
C01536=1044.684,308.048,386.662,172.225,40.750,157.798
C01537=1044.691,308.295,386.629,172.229,40.753,157.799
C01538=1044.698,308.543,386.596,172.233,40.755,157.800
C01539=1044.705,308.790,386.562,172.237,40.758,157.800
C01540=1044.711,309.037,386.529,172.240,40.761,157.801
C01541=1044.719,309.285,386.496,172.244,40.764,157.802
C01542=1044.726,309.533,386.462,172.248,40.766,157.803
C01543=1044.733,309.781,386.429,172.252,40.770,157.804
C01544=1044.740,310.028,386.396,172.256,40.772,157.804
C01545=1044.747,310.276,386.362,172.260,40.775,157.805
C01546=1044.754,310.523,386.328,172.264,40.777,157.806
C01547=1044.760,310.771,386.295,172.268,40.781,157.807
C01548=1044.768,311.019,386.261,172.272,40.783,157.808
C01549=1044.775,311.267,386.228,172.275,40.786,157.809
C01550=1044.781,311.514,386.194,172.279,40.789,157.809
C01551=1044.789,311.762,386.162,172.283,40.792,157.810
C01552=1044.796,312.009,386.128,172.287,40.794,157.811
C01553=1044.804,312.257,386.094,172.291,40.797,157.812
C01554=1044.811,312.505,386.060,172.295,40.800,157.813
C01555=1044.817,312.752,386.026,172.299,40.803,157.814
C01556=1044.824,313.000,385.992,172.303,40.806,157.814
C01557=1044.830,313.248,385.958,172.307,40.809,157.815
C01558=1044.837,313.495,385.924,172.311,40.812,157.816
C01559=1044.844,313.742,385.891,172.315,40.815,157.817
C01560=1044.850,313.990,385.856,172.319,40.818,157.818
C01561=1044.857,314.237,385.823,172.323,40.821,157.819
C01562=1044.864,314.485,385.788,172.327,40.824,157.820
C01563=1044.871,314.733,385.754,172.331,40.827,157.821
C01564=1044.878,314.980,385.719,172.335,40.830,157.821
C01565=1044.884,315.227,385.686,172.338,40.833,157.822
C01566=1044.891,315.475,385.651,172.342,40.836,157.823
C01567=1044.898,315.723,385.618,172.346,40.839,157.824
C01568=1044.904,315.971,385.583,172.350,40.842,157.825
C01569=1044.911,316.218,385.550,172.354,40.845,157.826
C01570=1044.918,316.465,385.515,172.358,40.848,157.827
C01571=1044.925,316.713,385.481,172.362,40.851,157.828
C01572=1044.931,316.961,385.446,172.366,40.854,157.828
C01573=1044.939,317.208,385.412,172.370,40.857,157.829
C01574=1044.945,317.455,385.378,172.374,40.860,157.830
C01575=1044.952,317.703,385.344,172.378,40.863,157.831
C01576=1044.958,317.951,385.310,172.382,40.866,157.832
C01577=1044.966,318.198,385.275,172.386,40.869,157.833
C01578=1044.972,318.446,385.241,172.390,40.872,157.834
C01579=1044.980,318.693,385.206,172.394,40.875,157.835
C01580=1044.988,319.017,385.161,172.399,40.880,157.836
C01581=1044.998,319.341,385.116,172.405,40.883,157.837
C01582=1045.007,319.664,385.071,172.410,40.888,157.838
C01583=1045.016,319.989,385.026,172.416,40.891,157.839
C01584=1045.023,320.236,384.992,172.420,40.894,157.840
C01585=1045.030,320.484,384.957,172.424,40.897,157.841
C01586=1045.037,320.731,384.923,172.428,40.901,157.842
C01587=1045.044,320.979,384.888,172.432,40.903,157.843
C01588=1045.050,321.227,384.853,172.436,40.907,157.844
C01589=1045.058,321.474,384.819,172.440,40.910,157.845
C01590=1045.064,321.722,384.784,172.445,40.913,157.846
C01591=1045.072,321.969,384.750,172.449,40.916,157.847
C01592=1045.078,322.216,384.715,172.453,40.919,157.848
C01593=1045.085,322.464,384.681,172.457,40.922,157.849
C01594=1045.092,322.711,384.646,172.461,40.925,157.849
C01595=1045.099,322.959,384.612,172.465,40.928,157.850
C01596=1045.106,323.206,384.577,172.470,40.931,157.851
C01597=1045.113,323.454,384.542,172.474,40.934,157.852
C01598=1045.121,323.701,384.507,172.478,40.938,157.853
C01599=1045.127,323.949,384.473,172.482,40.941,157.854
C01600=1045.134,324.196,384.438,172.486,40.944,157.855
C01601=1045.141,324.443,384.403,172.492,40.947,157.856
C01602=1045.149,324.691,384.368,172.496,40.950,157.857
C01603=1045.156,324.939,384.334,172.500,40.953,157.858
C01604=1045.163,325.186,384.298,172.504,40.957,157.859
C01605=1045.170,325.433,384.264,172.508,40.960,157.860
C01606=1045.177,325.681,384.229,172.513,40.963,157.861
C01607=1045.184,325.928,384.194,172.517,40.966,157.862
C01608=1045.192,326.176,384.159,172.521,40.969,157.863
C01609=1045.198,326.424,384.124,172.525,40.972,157.863
C01610=1045.206,326.671,384.090,172.530,40.976,157.864
C01611=1045.212,326.918,384.055,172.534,40.979,157.865
C01612=1045.221,327.166,384.020,172.538,40.982,157.866
C01613=1045.227,327.413,383.985,172.542,40.985,157.867
C01614=1045.234,327.661,383.949,172.547,40.988,157.868
C01615=1045.242,327.908,383.915,172.551,40.991,157.869
C01616=1045.249,328.156,383.879,172.555,40.995,157.870
C01617=1045.256,328.403,383.844,172.560,40.998,157.871
C01618=1045.263,328.650,383.810,172.564,41.001,157.872
C01619=1045.271,328.898,383.774,172.568,41.004,157.873
C01620=1045.278,329.145,383.740,172.573,41.008,157.874
C01621=1045.285,329.392,383.704,172.578,41.011,157.875
C01622=1045.293,329.640,383.668,172.582,41.014,157.876
C01623=1045.299,329.888,383.633,172.586,41.017,157.877
C01624=1045.306,330.135,383.598,172.591,41.021,157.878
C01625=1045.313,330.382,383.562,172.595,41.024,157.879
C01626=1045.321,330.630,383.527,172.599,41.027,157.880
C01627=1045.327,330.877,383.492,172.604,41.031,157.881
C01628=1045.334,331.124,383.456,172.608,41.034,157.882
C01629=1045.342,331.372,383.420,172.612,41.037,157.883
C01630=1045.349,331.619,383.385,172.617,41.041,157.884
C01631=1045.356,331.866,383.349,172.622,41.044,157.885
C01632=1045.363,332.114,383.314,172.626,41.048,157.886
C01633=1045.370,332.361,383.279,172.630,41.051,157.887
C01634=1045.377,332.608,383.243,172.635,41.054,157.888
C01635=1045.384,332.856,383.207,172.639,41.058,157.889
C01636=1045.393,333.175,383.161,172.645,41.062,157.890
C01637=1045.402,333.495,383.115,172.651,41.067,157.892
C01638=1045.412,333.813,383.069,172.657,41.071,157.893
C01639=1045.421,334.132,383.022,172.663,41.075,157.894
C01640=1045.428,334.380,382.987,172.667,41.079,157.895
C01641=1045.435,334.626,382.951,172.671,41.082,157.896
C01642=1045.442,334.874,382.915,172.676,41.085,157.897
C01643=1045.449,335.121,382.880,172.681,41.089,157.898
C01644=1045.457,335.369,382.844,172.685,41.092,157.899
C01645=1045.463,335.616,382.808,172.690,41.096,157.901
C01646=1045.471,335.863,382.772,172.694,41.099,157.901
C01647=1045.478,336.110,382.736,172.699,41.103,157.903
C01648=1045.485,336.358,382.700,172.704,41.106,157.904
C01649=1045.492,336.605,382.664,172.709,41.109,157.905
C01650=1045.500,336.853,382.628,172.713,41.113,157.906
C01651=1045.506,337.100,382.592,172.717,41.117,157.907
C01652=1045.514,337.347,382.556,172.722,41.120,157.908
C01653=1045.521,337.594,382.520,172.726,41.124,157.909
C01654=1045.528,337.841,382.483,172.732,41.127,157.910
C01655=1045.535,338.089,382.447,172.736,41.131,157.911
C01656=1045.542,338.336,382.411,172.741,41.135,157.912
C01657=1045.550,338.583,382.375,172.745,41.138,157.913
C01658=1045.556,338.831,382.339,172.749,41.142,157.914
C01659=1045.564,339.079,382.303,172.755,41.145,157.915
C01660=1045.571,339.326,382.266,172.759,41.149,157.916
C01661=1045.578,339.573,382.230,172.764,41.153,157.918
C01662=1045.586,339.820,382.193,172.768,41.156,157.919
C01663=1045.593,340.067,382.157,172.773,41.159,157.920
C01664=1045.600,340.314,382.120,172.778,41.163,157.921
C01665=1045.607,340.562,382.084,172.783,41.167,157.922
C01666=1045.615,340.809,382.048,172.787,41.170,157.923
C01667=1045.621,341.056,382.012,172.792,41.174,157.924
C01668=1045.629,341.304,381.975,172.797,41.178,157.925
C01669=1045.637,341.551,381.939,172.802,41.181,157.926
C01670=1045.643,341.798,381.902,172.806,41.185,157.927
C01671=1045.651,342.045,381.866,172.811,41.189,157.929
C01672=1045.659,342.293,381.829,172.817,41.192,157.930
C01673=1045.665,342.540,381.793,172.821,41.196,157.931
C01674=1045.673,342.786,381.756,172.826,41.200,157.932
C01675=1045.680,343.034,381.719,172.831,41.203,157.933
C01676=1045.687,343.282,381.682,172.836,41.207,157.934
C01677=1045.694,343.528,381.646,172.840,41.211,157.935
C01678=1045.701,343.776,381.609,172.845,41.215,157.936
C01679=1045.709,344.023,381.572,172.850,41.218,157.938
C01680=1045.716,344.270,381.535,172.855,41.222,157.939
C01681=1045.724,344.517,381.498,172.860,41.226,157.940
C01682=1045.731,344.764,381.462,172.864,41.229,157.941
C01683=1045.738,345.011,381.424,172.870,41.234,157.942
C01684=1045.745,345.259,381.388,172.874,41.237,157.943
C01685=1045.753,345.506,381.351,172.879,41.241,157.944
C01686=1045.760,345.753,381.315,172.885,41.244,157.946
C01687=1045.767,346.000,381.277,172.889,41.249,157.947
C01688=1045.774,346.248,381.241,172.894,41.252,157.948
C01689=1045.782,346.494,381.204,172.899,41.256,157.949
C01690=1045.789,346.742,381.166,172.904,41.260,157.950
C01691=1045.796,346.989,381.129,172.909,41.264,157.951
C01692=1045.805,347.275,381.087,172.915,41.268,157.953
C01693=1045.813,347.561,381.043,172.920,41.273,157.954
C01694=1045.822,347.847,381.001,172.926,41.277,157.956
C01695=1045.830,348.132,380.958,172.933,41.281,157.957
C01696=1045.837,348.380,380.920,172.937,41.286,157.958
C01697=1045.845,348.626,380.883,172.942,41.289,157.959
C01698=1045.853,348.874,380.846,172.948,41.293,157.961
C01699=1045.860,349.121,380.809,172.952,41.297,157.962
C01700=1045.868,349.368,380.772,172.957,41.301,157.963
C01701=1045.875,349.615,380.734,172.963,41.305,157.964
C01702=1045.882,349.862,380.697,172.967,41.309,157.965
C01703=1045.890,350.109,380.660,172.972,41.313,157.966
C01704=1045.897,350.356,380.622,172.978,41.317,157.968
C01705=1045.904,350.604,380.585,172.982,41.321,157.969
C01706=1045.912,350.851,380.547,172.988,41.325,157.970
C01707=1045.919,351.098,380.510,172.993,41.329,157.971
C01708=1045.927,351.346,380.472,172.998,41.332,157.973
C01709=1045.934,351.593,380.434,173.003,41.337,157.974
C01710=1045.942,351.839,380.396,173.008,41.341,157.975
C01711=1045.949,352.086,380.358,173.014,41.345,157.976
C01712=1045.956,352.334,380.321,173.019,41.349,157.977
C01713=1045.963,352.581,380.283,173.023,41.353,157.979
C01714=1045.971,352.828,380.247,173.029,41.357,157.980
C01715=1045.979,353.074,380.208,173.034,41.361,157.981
C01716=1045.986,353.321,380.171,173.040,41.365,157.983
C01717=1045.993,353.568,380.133,173.044,41.369,157.984
C01718=1046.001,353.815,380.095,173.050,41.373,157.985
C01719=1046.009,354.063,380.057,173.055,41.377,157.986
C01720=1046.016,354.310,380.020,173.061,41.381,157.988
C01721=1046.024,354.556,379.981,173.066,41.385,157.989
C01722=1046.031,354.803,379.944,173.070,41.390,157.990
C01723=1046.038,355.050,379.906,173.076,41.394,157.991
C01724=1046.046,355.298,379.868,173.081,41.398,157.993
C01725=1046.054,355.544,379.829,173.087,41.402,157.994
C01726=1046.061,355.791,379.792,173.092,41.406,157.995
C01727=1046.069,356.038,379.754,173.098,41.410,157.997
C01728=1046.076,356.286,379.716,173.102,41.415,157.998
C01729=1046.084,356.532,379.677,173.108,41.419,157.999
C01730=1046.091,356.779,379.640,173.113,41.423,158.000
C01731=1046.099,357.027,379.601,173.119,41.427,158.002
C01732=1046.107,357.273,379.563,173.124,41.431,158.003
C01733=1046.114,357.520,379.526,173.130,41.436,158.004
C01734=1046.121,357.767,379.487,173.135,41.440,158.006
C01735=1046.129,358.014,379.448,173.140,41.444,158.007
C01736=1046.136,358.261,379.411,173.145,41.448,158.008
C01737=1046.144,358.508,379.372,173.151,41.453,158.010
C01738=1046.152,358.755,379.334,173.156,41.457,158.011
C01739=1046.160,359.002,379.296,173.162,41.461,158.012
C01740=1046.166,359.249,379.257,173.168,41.466,158.014
C01741=1046.175,359.496,379.218,173.173,41.470,158.015
C01742=1046.182,359.742,379.180,173.179,41.474,158.016
C01743=1046.190,359.990,379.142,173.184,41.479,158.018
C01744=1046.197,360.237,379.104,173.190,41.483,158.019
C01745=1046.204,360.483,379.065,173.195,41.487,158.020
C01746=1046.212,360.731,379.026,173.201,41.492,158.022
C01747=1046.222,361.035,378.978,173.208,41.497,158.023
C01748=1046.234,361.415,378.919,173.216,41.503,158.026
C01749=1046.244,361.736,378.868,173.223,41.509,158.027
C01750=1046.254,362.056,378.819,173.230,41.515,158.029
C01751=1046.264,362.377,378.769,173.237,41.521,158.031
C01752=1046.271,362.625,378.730,173.243,41.525,158.032
C01753=1046.279,362.870,378.691,173.249,41.530,158.034
C01754=1046.287,363.118,378.652,173.254,41.535,158.035
C01755=1046.294,363.364,378.613,173.260,41.539,158.036
C01756=1046.303,363.611,378.574,173.266,41.543,158.038
C01757=1046.309,363.858,378.535,173.271,41.548,158.039
C01758=1046.317,364.105,378.496,173.277,41.553,158.041
C01759=1046.325,364.351,378.457,173.282,41.557,158.042
C01760=1046.333,364.599,378.418,173.288,41.561,158.044
C01761=1046.340,364.845,378.379,173.294,41.566,158.045
C01762=1046.347,365.092,378.339,173.299,41.571,158.046
C01763=1046.356,365.339,378.300,173.306,41.575,158.048
C01764=1046.363,365.586,378.261,173.312,41.580,158.049
C01765=1046.371,365.832,378.222,173.318,41.585,158.051
C01766=1046.378,366.080,378.183,173.323,41.589,158.052
C01767=1046.386,366.326,378.144,173.329,41.594,158.054
C01768=1046.394,366.573,378.105,173.335,41.598,158.055
C01769=1046.402,366.820,378.065,173.340,41.603,158.057
C01770=1046.409,367.066,378.026,173.346,41.608,158.058
C01771=1046.417,367.313,377.987,173.352,41.612,158.060
C01772=1046.425,367.560,377.947,173.357,41.617,158.061
C01773=1046.433,367.806,377.908,173.364,41.622,158.063
C01774=1046.441,368.053,377.868,173.370,41.626,158.064
C01775=1046.448,368.300,377.828,173.376,41.631,158.065
C01776=1046.457,368.547,377.790,173.381,41.635,158.067
C01777=1046.464,368.794,377.750,173.387,41.640,158.068
C01778=1046.472,369.040,377.711,173.393,41.645,158.070
C01779=1046.480,369.287,377.671,173.400,41.650,158.071
C01780=1046.488,369.533,377.632,173.405,41.654,158.073
C01781=1046.496,369.780,377.592,173.411,41.659,158.074
C01782=1046.505,370.027,377.552,173.417,41.664,158.076
C01783=1046.512,370.274,377.512,173.423,41.669,158.077
C01784=1046.519,370.520,377.473,173.429,41.673,158.079
C01785=1046.528,370.767,377.434,173.435,41.679,158.081
C01786=1046.536,371.013,377.394,173.441,41.683,158.082
C01787=1046.543,371.260,377.354,173.447,41.688,158.084
C01788=1046.552,371.507,377.314,173.454,41.693,158.085
C01789=1046.559,371.754,377.275,173.459,41.698,158.087
C01790=1046.567,372.000,377.234,173.465,41.703,158.088
C01791=1046.575,372.247,377.194,173.471,41.708,158.090
C01792=1046.583,372.494,377.154,173.478,41.712,158.091
C01793=1046.591,372.741,377.114,173.484,41.718,158.093
C01794=1046.598,372.986,377.074,173.490,41.723,158.095
C01795=1046.606,373.233,377.034,173.495,41.727,158.096
C01796=1046.614,373.480,376.993,173.502,41.732,158.098
C01797=1046.622,373.726,376.954,173.508,41.738,158.099
C01798=1046.630,373.973,376.914,173.514,41.743,158.101
C01799=1046.638,374.219,376.873,173.521,41.747,158.102
C01800=1046.646,374.466,376.834,173.527,41.752,158.104
C01801=1046.654,374.713,376.793,173.533,41.758,158.106
C01802=1046.661,374.960,376.753,173.540,41.763,158.107
C01803=1046.670,375.207,376.712,173.545,41.768,158.109
C01804=1046.681,375.546,376.656,173.554,41.774,158.111
C01805=1046.692,375.886,376.600,173.563,41.782,158.113
C01806=1046.703,376.226,376.545,173.571,41.789,158.116
C01807=1046.714,376.567,376.490,173.580,41.796,158.118
C01808=1046.722,376.813,376.449,173.587,41.801,158.120
C01809=1046.730,377.059,376.409,173.593,41.806,158.121
C01810=1046.739,377.306,376.368,173.599,41.811,158.123
C01811=1046.747,377.553,376.327,173.606,41.816,158.124
C01812=1046.755,377.799,376.287,173.612,41.822,158.126
C01813=1046.763,378.046,376.246,173.619,41.827,158.128
C01814=1046.771,378.293,376.205,173.625,41.832,158.129
C01815=1046.779,378.539,376.165,173.632,41.837,158.131
C01816=1046.787,378.785,376.124,173.638,41.842,158.133
C01817=1046.795,379.032,376.083,173.645,41.847,158.135
C01818=1046.804,379.279,376.042,173.651,41.853,158.136
